LIN {X 0,Y 539.929,Z 932.451,A -85,B 0,C 180,E1 4064.865,E2 4064.865} C_VEL
LIN {X 0,Y 540.898,Z 908.583,A -85,B 0,C 180,E1 4068.356,E2 4068.356} C_VEL
LIN {X 0,Y 542.169,Z 880.394,A -85,B 0,C 180,E1 4071.395,E2 4071.395} C_VEL
LIN {X 0,Y 543.664,Z 848.735,A -85,B 0,C 180,E1 4073.926,E2 4073.926} C_VEL
LIN {X 0,Y 545.192,Z 813.47,A -85,B 0,C 180,E1 4075.928,E2 4075.928} C_VEL
LIN {X 0,Y 546.363,Z 778.099,A -85,B 0,C 180,E1 4077.245,E2 4077.245} C_VEL
LIN {X 0,Y 546.243,Z 753.317,A -85,B 0,C 180,E1 4077.845,E2 4077.845} C_VEL
LIN {X 0,Y 538.505,Z 733.66,A -85,B 0,C 180,E1 4078.65,E2 4078.65} C_VEL
LIN {X 0,Y 538.24,Z 733.66,A -85,B 0,C 180,E1 4084.237,E2 4084.237} C_VEL
LIN {X 0,Y 538.141,Z 733.66,A -85,B 0,C 180,E1 4090.325,E2 4090.325} C_VEL
LIN {X 0,Y 538.198,Z 733.66,A -85,B 0,C 180,E1 4095.304,E2 4095.304} C_VEL
LIN {X 0,Y 538.244,Z 733.66,A -85,B 0,C 180,E1 4101.765,E2 4101.765} C_VEL
LIN {X 0,Y 538.178,Z 733.66,A -85,B 0,C 180,E1 4107.685,E2 4107.685} C_VEL
LIN {X 0,Y 538.392,Z 733.66,A -85,B 0,C 180,E1 4113.256,E2 4113.256} C_VEL
LIN {X 0,Y 538.489,Z 733.66,A -85,B 0,C 180,E1 4118.557,E2 4118.557} C_VEL
LIN {X 0,Y 538.505,Z 733.66,A -85,B 0,C 180,E1 4123.667,E2 4123.667} C_VEL
LIN {X 0,Y 538.551,Z 733.66,A -85,B 0,C 180,E1 4130.286,E2 4130.286} C_VEL
LIN {X 0,Y 538.695,Z 733.66,A -85,B 0,C 180,E1 4135.16,E2 4135.16} C_VEL
LIN {X 0,Y 538.731,Z 733.66,A -85,B 0,C 180,E1 4139.996,E2 4139.996} C_VEL
LIN {X 0,Y 538.698,Z 733.66,A -85,B 0,C 180,E1 4144.833,E2 4144.833} C_VEL
LIN {X 0,Y 538.561,Z 733.66,A -85,B 0,C 180,E1 4150.268,E2 4150.268} C_VEL
LIN {X 0,Y 538.552,Z 733.66,A -85,B 0,C 180,E1 4154.652,E2 4154.652} C_VEL
LIN {X 0,Y 538.526,Z 733.66,A -85,B 0,C 180,E1 4159.713,E2 4159.713} C_VEL
LIN {X 0,Y 538.328,Z 733.66,A -85,B 0,C 180,E1 4165.302,E2 4165.302} C_VEL
LIN {X 0,Y 537.026,Z 733.66,A -85,B 0,C 180,E1 4166.225,E2 4166.225} C_VEL
LIN {X 0,Y 530.436,Z 733.66,A -85,B 0,C 180,E1 4168.737,E2 4168.737} C_VEL
LIN {X 0,Y 530.367,Z 733.66,A -85,B 0,C 180,E1 4168.975,E2 4168.975} C_VEL
LIN {X 0,Y 530.295,Z 733.66,A -85,B 0,C 180,E1 4174.816,E2 4174.816} C_VEL
LIN {X 0,Y 530.19,Z 733.66,A -85,B 0,C 180,E1 4181.05,E2 4181.05} C_VEL
LIN {X 0,Y 530.337,Z 733.66,A -85,B 0,C 180,E1 4186.749,E2 4186.749} C_VEL
LIN {X 0,Y 530.299,Z 733.66,A -85,B 0,C 180,E1 4193.067,E2 4193.067} C_VEL
LIN {X 0,Y 530.392,Z 734.199,A -85,B 0,C 180,E1 4198.178,E2 4198.178} C_VEL
LIN {X 0,Y 534.911,Z 747.208,A -85,B 0,C 180,E1 4199.252,E2 4199.252} C_VEL
LIN {X 0,Y 543.352,Z 759.578,A -85,B 0,C 180,E1 4200.686,E2 4200.686} C_VEL
LIN {X 0,Y 540.185,Z 771.164,A -85,B 0,C 180,E1 4201.27,E2 4201.27} C_VEL
LIN {X 0,Y 539.525,Z 822.398,A -85,B 0,C 180,E1 4202.164,E2 4202.164} C_VEL
LIN {X 0,Y 538.205,Z 858.389,A -85,B 0,C 180,E1 4203.418,E2 4203.418} C_VEL
LIN {X 0,Y 536.657,Z 892.998,A -85,B 0,C 180,E1 4205.297,E2 4205.297} C_VEL
LIN {X 0,Y 534.865,Z 926.522,A -85,B 0,C 180,E1 4207.881,E2 4207.881} C_VEL
LIN {X 0,Y 533.463,Z 953.726,A -85,B 0,C 180,E1 4210.734,E2 4210.734} C_VEL
LIN {X 0,Y 532.298,Z 977.994,A -85,B 0,C 180,E1 4214.111,E2 4214.111} C_VEL
LIN {X 0,Y 531.607,Z 996.677,A -85,B 0,C 180,E1 4217.666,E2 4217.666} C_VEL
LIN {X 0,Y 531.266,Z 1010.424,A -85,B 0,C 180,E1 4221.395,E2 4221.395} C_VEL
LIN {X 0,Y 531.098,Z 1018.952,A -85,B 0,C 180,E1 4225.093,E2 4225.093} C_VEL
LIN {X 0,Y 531.029,Z 1022.53,A -85,B 0,C 180,E1 4228.366,E2 4228.366} C_VEL
LIN {X 0,Y 531.093,Z 1022.529,A -85,B 0,C 180,E1 4231.633,E2 4231.633} C_VEL
LIN {X 0,Y 531.095,Z 1017.469,A -85,B 0,C 180,E1 4235.726,E2 4235.726} C_VEL
LIN {X 0,Y 531.28,Z 1007.861,A -85,B 0,C 180,E1 4239.431,E2 4239.431} C_VEL
LIN {X 0,Y 531.693,Z 992.833,A -85,B 0,C 180,E1 4243.168,E2 4243.168} C_VEL
LIN {X 0,Y 532.477,Z 971.655,A -85,B 0,C 180,E1 4246.872,E2 4246.872} C_VEL
LIN {X 0,Y 533.771,Z 946.485,A -85,B 0,C 180,E1 4250.107,E2 4250.107} C_VEL
LIN {X 0,Y 535.394,Z 917.124,A -85,B 0,C 180,E1 4252.931,E2 4252.931} C_VEL
LIN {X 0,Y 537.131,Z 884.48,A -85,B 0,C 180,E1 4255.23,E2 4255.23} C_VEL
LIN {X 0,Y 538.607,Z 850.059,A -85,B 0,C 180,E1 4256.929,E2 4256.929} C_VEL
LIN {X 0,Y 539.757,Z 813.547,A -85,B 0,C 180,E1 4258.047,E2 4258.047} C_VEL
LIN {X 0,Y 540.347,Z 770.37,A -85,B 0,C 180,E1 4258.776,E2 4258.776} C_VEL
LIN {X 0,Y 543.301,Z 759.584,A -85,B 0,C 180,E1 4259.319,E2 4259.319} C_VEL
LIN {X 0,Y 535.922,Z 748.545,A -85,B 0,C 180,E1 4260.605,E2 4260.605} C_VEL
LIN {X 0,Y 531.135,Z 737.856,A -85,B 0,C 180,E1 4261.416,E2 4261.416} C_VEL
LIN {X 0,Y 530.394,Z 733.66,A -85,B 0,C 180,E1 4261.772,E2 4261.772} C_VEL
LIN {X 0,Y 530.271,Z 733.66,A -85,B 0,C 180,E1 4266.929,E2 4266.929} C_VEL
LIN {X 0,Y 530.332,Z 733.66,A -85,B 0,C 180,E1 4273.251,E2 4273.251} C_VEL
LIN {X 0,Y 530.202,Z 733.66,A -85,B 0,C 180,E1 4278.951,E2 4278.951} C_VEL
LIN {X 0,Y 530.313,Z 733.66,A -85,B 0,C 180,E1 4285.185,E2 4285.185} C_VEL
LIN {X 0,Y 530.38,Z 733.66,A -85,B 0,C 180,E1 4290.974,E2 4290.974} C_VEL
LIN {X 0,Y 530.358,Z 733.66,A -85,B 0,C 180,E1 4296.447,E2 4296.447} C_VEL
LIN {X 0,Y 530.588,Z 733.66,A -85,B 0,C 180,E1 4299.925,E2 4299.925} C_VEL
LIN {X 0,Y 534.239,Z 751.767,A -85,B 0,C 180,E1 4300.375,E2 4300.375} C_VEL
LIN {X 0,Y 534.049,Z 781.281,A -85,B 0,C 180,E1 4301.36,E2 4301.36} C_VEL
LIN {X 0,Y 533.37,Z 807.505,A -85,B 0,C 180,E1 4302.911,E2 4302.911} C_VEL
LIN {X 0,Y 532.655,Z 830.205,A -85,B 0,C 180,E1 4304.993,E2 4304.993} C_VEL
LIN {X 0,Y 532.005,Z 848.565,A -85,B 0,C 180,E1 4307.471,E2 4307.471} C_VEL
LIN {X 0,Y 531.572,Z 861.83,A -85,B 0,C 180,E1 4310.164,E2 4310.164} C_VEL
LIN {X 0,Y 531.368,Z 871.236,A -85,B 0,C 180,E1 4313.459,E2 4313.459} C_VEL
LIN {X 0,Y 531.216,Z 874.4,A -85,B 0,C 180,E1 4316.736,E2 4316.736} C_VEL
LIN {X 0,Y 531.291,Z 871.871,A -85,B 0,C 180,E1 4320.004,E2 4320.004} C_VEL
LIN {X 0,Y 531.451,Z 864.702,A -85,B 0,C 180,E1 4322.861,E2 4322.861} C_VEL
LIN {X 0,Y 531.852,Z 850.948,A -85,B 0,C 180,E1 4325.927,E2 4325.927} C_VEL
LIN {X 0,Y 532.375,Z 832.207,A -85,B 0,C 180,E1 4328.59,E2 4328.59} C_VEL
LIN {X 0,Y 533.103,Z 809.618,A -85,B 0,C 180,E1 4330.745,E2 4330.745} C_VEL
LIN {X 0,Y 533.865,Z 783.985,A -85,B 0,C 180,E1 4332.354,E2 4332.354} C_VEL
LIN {X 0,Y 534.405,Z 755.268,A -85,B 0,C 180,E1 4333.417,E2 4333.417} C_VEL
LIN {X 0,Y 532.781,Z 741.992,A -85,B 0,C 180,E1 4333.748,E2 4333.748} C_VEL
LIN {X 0,Y 530.642,Z 733.66,A -85,B 0,C 180,E1 4334.04,E2 4334.04} C_VEL
LIN {X 0,Y 530.553,Z 733.66,A -85,B 0,C 180,E1 4340.029,E2 4340.029} C_VEL
LIN {X 0,Y 530.431,Z 733.66,A -85,B 0,C 180,E1 4345.354,E2 4345.354} C_VEL
LIN {X 0,Y 530.297,Z 733.66,A -85,B 0,C 180,E1 4351.069,E2 4351.069} C_VEL
LIN {X 0,Y 530.234,Z 733.66,A -85,B 0,C 180,E1 4356.914,E2 4356.914} C_VEL
LIN {X 0,Y 530.302,Z 733.66,A -85,B 0,C 180,E1 4363.256,E2 4363.256} C_VEL
LIN {X 0,Y 530.31,Z 733.66,A -85,B 0,C 180,E1 4368.954,E2 4368.954} C_VEL
LIN {X 0,Y 530.286,Z 733.66,A -85,B 0,C 180,E1 4375.177,E2 4375.177} C_VEL
LIN {X 0,Y 530.42,Z 733.66,A -85,B 0,C 180,E1 4380.828,E2 4380.828} C_VEL
LIN {X 0,Y 539.68,Z 758.857,A -85,B 0,C 180,E1 4381.801,E2 4381.801} C_VEL
LIN {X 0,Y 538.677,Z 797.066,A -85,B 0,C 180,E1 4382.911,E2 4382.911} C_VEL
LIN {X 0,Y 537.216,Z 832.111,A -85,B 0,C 180,E1 4384.59,E2 4384.59} C_VEL
LIN {X 0,Y 535.516,Z 864.375,A -85,B 0,C 180,E1 4386.8,E2 4386.8} C_VEL
LIN {X 0,Y 533.886,Z 895.221,A -85,B 0,C 180,E1 4389.706,E2 4389.706} C_VEL
LIN {X 0,Y 532.582,Z 920.869,A -85,B 0,C 180,E1 4392.968,E2 4392.968} C_VEL
LIN {X 0,Y 531.851,Z 941.307,A -85,B 0,C 180,E1 4396.474,E2 4396.474} C_VEL
LIN {X 0,Y 531.367,Z 956.651,A -85,B 0,C 180,E1 4400.156,E2 4400.156} C_VEL
LIN {X 0,Y 531.192,Z 965.865,A -85,B 0,C 180,E1 4403.453,E2 4403.453} C_VEL
LIN {X 0,Y 531.107,Z 971.214,A -85,B 0,C 180,E1 4406.732,E2 4406.732} C_VEL
LIN {X 0,Y 531.074,Z 972.997,A -85,B 0,C 180,E1 4410,E2 4410} C_VEL
LIN {X 0,Y 531.156,Z 970.398,A -85,B 0,C 180,E1 4413.883,E2 4413.883} C_VEL
LIN {X 0,Y 531.252,Z 962.625,A -85,B 0,C 180,E1 4417.781,E2 4417.781} C_VEL
LIN {X 0,Y 531.478,Z 950.035,A -85,B 0,C 180,E1 4421.503,E2 4421.503} C_VEL
LIN {X 0,Y 532.216,Z 931.471,A -85,B 0,C 180,E1 4425.257,E2 4425.257} C_VEL
LIN {X 0,Y 533.292,Z 906.861,A -85,B 0,C 180,E1 4428.842,E2 4428.842} C_VEL
LIN {X 0,Y 534.784,Z 878.331,A -85,B 0,C 180,E1 4431.905,E2 4431.905} C_VEL
LIN {X 0,Y 536.522,Z 845.585,A -85,B 0,C 180,E1 4434.487,E2 4434.487} C_VEL
LIN {X 0,Y 538.09,Z 813.068,A -85,B 0,C 180,E1 4436.316,E2 4436.316} C_VEL
LIN {X 0,Y 539.356,Z 778.111,A -85,B 0,C 180,E1 4437.629,E2 4437.629} C_VEL
LIN {X 0,Y 539.212,Z 755.599,A -85,B 0,C 180,E1 4438.198,E2 4438.198} C_VEL
LIN {X 0,Y 530.524,Z 733.66,A -85,B 0,C 180,E1 4439.114,E2 4439.114} C_VEL
LIN {X 0,Y 530.312,Z 733.66,A -85,B 0,C 180,E1 4444.822,E2 4444.822} C_VEL
LIN {X 0,Y 530.193,Z 733.66,A -85,B 0,C 180,E1 4451.058,E2 4451.058} C_VEL
LIN {X 0,Y 530.318,Z 733.66,A -85,B 0,C 180,E1 4456.745,E2 4456.745} C_VEL
LIN {X 0,Y 530.267,Z 733.66,A -85,B 0,C 180,E1 4463.155,E2 4463.155} C_VEL
LIN {X 0,Y 530.274,Z 733.66,A -85,B 0,C 180,E1 4469.07,E2 4469.07} C_VEL
LIN {X 0,Y 530.512,Z 733.66,A -85,B 0,C 180,E1 4474.65,E2 4474.65} C_VEL
LIN {X 0,Y 530.696,Z 733.66,A -85,B 0,C 180,E1 4480.306,E2 4480.306} C_VEL
LIN {X 0,Y 530.363,Z 733.66,A -85,B 0,C 180,E1 4486.083,E2 4486.083} C_VEL
LIN {X 0,Y 530.653,Z 733.66,A -85,B 0,C 180,E1 4491.795,E2 4491.795} C_VEL
LIN {X 0,Y 530.732,Z 733.66,A -85,B 0,C 180,E1 4496.86,E2 4496.86} C_VEL
LIN {X 0,Y 530.746,Z 733.66,A -85,B 0,C 180,E1 4501.631,E2 4501.631} C_VEL
LIN {X 0,Y 530.702,Z 733.66,A -85,B 0,C 180,E1 4506.549,E2 4506.549} C_VEL
LIN {X 0,Y 530.651,Z 733.66,A -85,B 0,C 180,E1 4511.517,E2 4511.517} C_VEL
LIN {X 0,Y 530.598,Z 733.66,A -85,B 0,C 180,E1 4516.575,E2 4516.575} C_VEL
LIN {X 0,Y 530.538,Z 733.66,A -85,B 0,C 180,E1 4521.772,E2 4521.772} C_VEL
LIN {X 0,Y 530.358,Z 733.66,A -85,B 0,C 180,E1 4527.747,E2 4527.747} C_VEL
LIN {X 0,Y 530.367,Z 733.66,A -85,B 0,C 180,E1 4528.975,E2 4528.975} C_VEL
LIN {X 0,Y 527.852,Z 733.66,A -85,B 0,C 180,E1 4530.369,E2 4530.369} C_VEL
LIN {X 0,Y 522.463,Z 733.66,A -85,B 0,C 180,E1 4532.458,E2 4532.458} C_VEL
LIN {X 0,Y 522.395,Z 733.66,A -85,B 0,C 180,E1 4532.699,E2 4532.699} C_VEL
LIN {X 0,Y 522.248,Z 733.66,A -85,B 0,C 180,E1 4538.484,E2 4538.484} C_VEL
LIN {X 0,Y 522.388,Z 733.66,A -85,B 0,C 180,E1 4544.068,E2 4544.068} C_VEL
LIN {X 0,Y 522.41,Z 733.66,A -85,B 0,C 180,E1 4550.385,E2 4550.385} C_VEL
LIN {X 0,Y 522.363,Z 733.66,A -85,B 0,C 180,E1 4556.583,E2 4556.583} C_VEL
LIN {X 0,Y 522.469,Z 734.17,A -85,B 0,C 180,E1 4557.761,E2 4557.761} C_VEL
LIN {X 0,Y 528.528,Z 751.834,A -85,B 0,C 180,E1 4559.239,E2 4559.239} C_VEL
LIN {X 0,Y 536.281,Z 762.43,A -85,B 0,C 180,E1 4560.311,E2 4560.311} C_VEL
LIN {X 0,Y 533.224,Z 774.555,A -85,B 0,C 180,E1 4560.915,E2 4560.915} C_VEL
LIN {X 0,Y 532.534,Z 822.756,A -85,B 0,C 180,E1 4561.776,E2 4561.776} C_VEL
LIN {X 0,Y 531.071,Z 859.288,A -85,B 0,C 180,E1 4563.075,E2 4563.075} C_VEL
LIN {X 0,Y 529.28,Z 894.607,A -85,B 0,C 180,E1 4565.042,E2 4565.042} C_VEL
LIN {X 0,Y 527.318,Z 927.968,A -85,B 0,C 180,E1 4567.683,E2 4567.683} C_VEL
LIN {X 0,Y 525.636,Z 957.199,A -85,B 0,C 180,E1 4570.873,E2 4570.873} C_VEL
LIN {X 0,Y 524.433,Z 980.46,A -85,B 0,C 180,E1 4574.296,E2 4574.296} C_VEL
LIN {X 0,Y 523.674,Z 998.511,A -85,B 0,C 180,E1 4577.9,E2 4577.9} C_VEL
LIN {X 0,Y 523.342,Z 1011.603,A -85,B 0,C 180,E1 4581.682,E2 4581.682} C_VEL
LIN {X 0,Y 523.201,Z 1018.949,A -85,B 0,C 180,E1 4585.019,E2 4585.019} C_VEL
LIN {X 0,Y 523.144,Z 1022.532,A -85,B 0,C 180,E1 4588.341,E2 4588.341} C_VEL
LIN {X 0,Y 523.204,Z 1022.531,A -85,B 0,C 180,E1 4591.658,E2 4591.658} C_VEL
LIN {X 0,Y 523.21,Z 1017.471,A -85,B 0,C 180,E1 4595.813,E2 4595.813} C_VEL
LIN {X 0,Y 523.411,Z 1007.857,A -85,B 0,C 180,E1 4599.574,E2 4599.574} C_VEL
LIN {X 0,Y 523.869,Z 992.835,A -85,B 0,C 180,E1 4603.368,E2 4603.368} C_VEL
LIN {X 0,Y 524.758,Z 972.047,A -85,B 0,C 180,E1 4607.066,E2 4607.066} C_VEL
LIN {X 0,Y 526.17,Z 946.886,A -85,B 0,C 180,E1 4610.364,E2 4610.364} C_VEL
LIN {X 0,Y 528.004,Z 917.072,A -85,B 0,C 180,E1 4613.275,E2 4613.275} C_VEL
LIN {X 0,Y 529.888,Z 884.475,A -85,B 0,C 180,E1 4615.6,E2 4615.6} C_VEL
LIN {X 0,Y 531.544,Z 849.967,A -85,B 0,C 180,E1 4617.32,E2 4617.32} C_VEL
LIN {X 0,Y 532.802,Z 813.504,A -85,B 0,C 180,E1 4618.448,E2 4618.448} C_VEL
LIN {X 0,Y 533.558,Z 772.405,A -85,B 0,C 180,E1 4619.177,E2 4619.177} C_VEL
LIN {X 0,Y 535.699,Z 761.602,A -85,B 0,C 180,E1 4619.779,E2 4619.779} C_VEL
LIN {X 0,Y 525.526,Z 746.23,A -85,B 0,C 180,E1 4621.098,E2 4621.098} C_VEL
LIN {X 0,Y 522.474,Z 733.66,A -85,B 0,C 180,E1 4622.031,E2 4622.031} C_VEL
LIN {X 0,Y 522.332,Z 733.66,A -85,B 0,C 180,E1 4628.506,E2 4628.506} C_VEL
LIN {X 0,Y 522.41,Z 733.66,A -85,B 0,C 180,E1 4634.074,E2 4634.074} C_VEL
LIN {X 0,Y 522.299,Z 733.66,A -85,B 0,C 180,E1 4640.383,E2 4640.383} C_VEL
LIN {X 0,Y 522.441,Z 733.66,A -85,B 0,C 180,E1 4646.596,E2 4646.596} C_VEL
LIN {X 0,Y 522.393,Z 733.66,A -85,B 0,C 180,E1 4652.377,E2 4652.377} C_VEL
LIN {X 0,Y 522.501,Z 733.66,A -85,B 0,C 180,E1 4658.016,E2 4658.016} C_VEL
LIN {X 0,Y 522.642,Z 734.005,A -85,B 0,C 180,E1 4659.662,E2 4659.662} C_VEL
LIN {X 0,Y 526.784,Z 753.759,A -85,B 0,C 180,E1 4660.154,E2 4660.154} C_VEL
LIN {X 0,Y 526.518,Z 782.775,A -85,B 0,C 180,E1 4661.142,E2 4661.142} C_VEL
LIN {X 0,Y 525.827,Z 808.359,A -85,B 0,C 180,E1 4662.67,E2 4662.67} C_VEL
LIN {X 0,Y 525.1,Z 830.995,A -85,B 0,C 180,E1 4664.75,E2 4664.75} C_VEL
LIN {X 0,Y 524.365,Z 849.627,A -85,B 0,C 180,E1 4667.285,E2 4667.285} C_VEL
LIN {X 0,Y 523.869,Z 862.972,A -85,B 0,C 180,E1 4670.018,E2 4670.018} C_VEL
LIN {X 0,Y 523.711,Z 870.701,A -85,B 0,C 180,E1 4672.529,E2 4672.529} C_VEL
LIN {X 0,Y 523.586,Z 874.779,A -85,B 0,C 180,E1 4675.027,E2 4675.027} C_VEL
LIN {X 0,Y 523.461,Z 875.097,A -85,B 0,C 180,E1 4678.346,E2 4678.346} C_VEL
LIN {X 0,Y 523.546,Z 869.653,A -85,B 0,C 180,E1 4681.661,E2 4681.661} C_VEL
LIN {X 0,Y 523.874,Z 859.139,A -85,B 0,C 180,E1 4684.648,E2 4684.648} C_VEL
LIN {X 0,Y 524.375,Z 843.193,A -85,B 0,C 180,E1 4687.469,E2 4687.469} C_VEL
LIN {X 0,Y 525.111,Z 821.857,A -85,B 0,C 180,E1 4689.966,E2 4689.966} C_VEL
LIN {X 0,Y 525.957,Z 796.971,A -85,B 0,C 180,E1 4691.901,E2 4691.901} C_VEL
LIN {X 0,Y 526.575,Z 769.577,A -85,B 0,C 180,E1 4693.244,E2 4693.244} C_VEL
LIN {X 0,Y 526.194,Z 746.991,A -85,B 0,C 180,E1 4693.888,E2 4693.888} C_VEL
LIN {X 0,Y 522.705,Z 733.66,A -85,B 0,C 180,E1 4694.258,E2 4694.258} C_VEL
LIN {X 0,Y 522.614,Z 733.66,A -85,B 0,C 180,E1 4700.347,E2 4700.347} C_VEL
LIN {X 0,Y 522.434,Z 733.66,A -85,B 0,C 180,E1 4706.048,E2 4706.048} C_VEL
LIN {X 0,Y 522.367,Z 733.66,A -85,B 0,C 180,E1 4711.451,E2 4711.451} C_VEL
LIN {X 0,Y 522.277,Z 733.66,A -85,B 0,C 180,E1 4717.505,E2 4717.505} C_VEL
LIN {X 0,Y 522.382,Z 733.66,A -85,B 0,C 180,E1 4723.564,E2 4723.564} C_VEL
LIN {X 0,Y 522.436,Z 733.66,A -85,B 0,C 180,E1 4728.898,E2 4728.898} C_VEL
LIN {X 0,Y 522.316,Z 733.66,A -85,B 0,C 180,E1 4734.567,E2 4734.567} C_VEL
LIN {X 0,Y 522.472,Z 733.66,A -85,B 0,C 180,E1 4740.322,E2 4740.322} C_VEL
LIN {X 0,Y 532.696,Z 761.121,A -85,B 0,C 180,E1 4741.446,E2 4741.446} C_VEL
LIN {X 0,Y 531.529,Z 799.009,A -85,B 0,C 180,E1 4742.6,E2 4742.6} C_VEL
LIN {X 0,Y 529.903,Z 833.765,A -85,B 0,C 180,E1 4744.316,E2 4744.316} C_VEL
LIN {X 0,Y 527.982,Z 866.735,A -85,B 0,C 180,E1 4746.647,E2 4746.647} C_VEL
LIN {X 0,Y 526.281,Z 895.955,A -85,B 0,C 180,E1 4749.485,E2 4749.485} C_VEL
LIN {X 0,Y 524.901,Z 920.495,A -85,B 0,C 180,E1 4752.656,E2 4752.656} C_VEL
LIN {X 0,Y 524.042,Z 941.496,A -85,B 0,C 180,E1 4756.307,E2 4756.307} C_VEL
LIN {X 0,Y 523.496,Z 956.649,A -85,B 0,C 180,E1 4760.007,E2 4760.007} C_VEL
LIN {X 0,Y 523.293,Z 965.864,A -85,B 0,C 180,E1 4763.354,E2 4763.354} C_VEL
LIN {X 0,Y 523.219,Z 971.213,A -85,B 0,C 180,E1 4766.682,E2 4766.682} C_VEL
LIN {X 0,Y 523.184,Z 972.997,A -85,B 0,C 180,E1 4770,E2 4770} C_VEL
LIN {X 0,Y 523.248,Z 970.399,A -85,B 0,C 180,E1 4773.942,E2 4773.942} C_VEL
LIN {X 0,Y 523.364,Z 962.627,A -85,B 0,C 180,E1 4777.899,E2 4777.899} C_VEL
LIN {X 0,Y 523.612,Z 950.036,A -85,B 0,C 180,E1 4781.678,E2 4781.678} C_VEL
LIN {X 0,Y 524.414,Z 931.478,A -85,B 0,C 180,E1 4785.49,E2 4785.49} C_VEL
LIN {X 0,Y 525.662,Z 906.864,A -85,B 0,C 180,E1 4789.126,E2 4789.126} C_VEL
LIN {X 0,Y 527.234,Z 879.552,A -85,B 0,C 180,E1 4792.116,E2 4792.116} C_VEL
LIN {X 0,Y 529.145,Z 847.228,A -85,B 0,C 180,E1 4794.739,E2 4794.739} C_VEL
LIN {X 0,Y 530.988,Z 813.08,A -85,B 0,C 180,E1 4796.695,E2 4796.695} C_VEL
LIN {X 0,Y 532.325,Z 778.628,A -85,B 0,C 180,E1 4798.01,E2 4798.01} C_VEL
LIN {X 0,Y 532.064,Z 757.239,A -85,B 0,C 180,E1 4798.58,E2 4798.58} C_VEL
LIN {X 0,Y 522.551,Z 733.66,A -85,B 0,C 180,E1 4799.626,E2 4799.626} C_VEL
LIN {X 0,Y 522.315,Z 733.66,A -85,B 0,C 180,E1 4805.739,E2 4805.739} C_VEL
LIN {X 0,Y 522.303,Z 733.66,A -85,B 0,C 180,E1 4811.816,E2 4811.816} C_VEL
LIN {X 0,Y 522.371,Z 733.66,A -85,B 0,C 180,E1 4818.188,E2 4818.188} C_VEL
LIN {X 0,Y 522.302,Z 733.66,A -85,B 0,C 180,E1 4824.563,E2 4824.563} C_VEL
LIN {X 0,Y 522.375,Z 733.66,A -85,B 0,C 180,E1 4830.477,E2 4830.477} C_VEL
LIN {X 0,Y 522.594,Z 733.66,A -85,B 0,C 180,E1 4836.068,E2 4836.068} C_VEL
LIN {X 0,Y 522.74,Z 733.66,A -85,B 0,C 180,E1 4841.418,E2 4841.418} C_VEL
LIN {X 0,Y 522.626,Z 733.66,A -85,B 0,C 180,E1 4848.296,E2 4848.296} C_VEL
LIN {X 0,Y 522.94,Z 733.66,A -85,B 0,C 180,E1 4853.346,E2 4853.346} C_VEL
LIN {X 0,Y 522.949,Z 733.66,A -85,B 0,C 180,E1 4859.996,E2 4859.996} C_VEL
LIN {X 0,Y 522.87,Z 733.66,A -85,B 0,C 180,E1 4864.98,E2 4864.98} C_VEL
LIN {X 0,Y 522.808,Z 733.66,A -85,B 0,C 180,E1 4870.045,E2 4870.045} C_VEL
LIN {X 0,Y 522.703,Z 733.66,A -85,B 0,C 180,E1 4875.107,E2 4875.107} C_VEL
LIN {X 0,Y 522.632,Z 733.66,A -85,B 0,C 180,E1 4880.338,E2 4880.338} C_VEL
LIN {X 0,Y 522.463,Z 733.66,A -85,B 0,C 180,E1 4886.054,E2 4886.054} C_VEL
LIN {X 0,Y 522.369,Z 733.66,A -85,B 0,C 180,E1 4891.442,E2 4891.442} C_VEL
LIN {X 0,Y 522.395,Z 733.66,A -85,B 0,C 180,E1 4892.699,E2 4892.699} C_VEL
LIN {X 0,Y 519.924,Z 733.66,A -85,B 0,C 180,E1 4894.111,E2 4894.111} C_VEL
LIN {X 0,Y 514.447,Z 733.66,A -85,B 0,C 180,E1 4896.226,E2 4896.226} C_VEL
LIN {X 0,Y 514.339,Z 733.66,A -85,B 0,C 180,E1 4896.471,E2 4896.471} C_VEL
LIN {X 0,Y 514.412,Z 733.66,A -85,B 0,C 180,E1 4902.622,E2 4902.622} C_VEL
LIN {X 0,Y 514.482,Z 733.66,A -85,B 0,C 180,E1 4907.4,E2 4907.4} C_VEL
LIN {X 0,Y 514.453,Z 733.66,A -85,B 0,C 180,E1 4912.611,E2 4912.611} C_VEL
LIN {X 0,Y 514.499,Z 733.748,A -85,B 0,C 180,E1 4917.299,E2 4917.299} C_VEL
LIN {X 0,Y 521.232,Z 755.025,A -85,B 0,C 180,E1 4919.085,E2 4919.085} C_VEL
LIN {X 0,Y 528.098,Z 766.006,A -85,B 0,C 180,E1 4920.141,E2 4920.141} C_VEL
LIN {X 0,Y 526.137,Z 775.03,A -85,B 0,C 180,E1 4920.548,E2 4920.548} C_VEL
LIN {X 0,Y 525.43,Z 822.995,A -85,B 0,C 180,E1 4921.403,E2 4921.403} C_VEL
LIN {X 0,Y 523.929,Z 860.182,A -85,B 0,C 180,E1 4922.723,E2 4922.723} C_VEL
LIN {X 0,Y 521.922,Z 896.215,A -85,B 0,C 180,E1 4924.78,E2 4924.78} C_VEL
LIN {X 0,Y 519.855,Z 928.496,A -85,B 0,C 180,E1 4927.396,E2 4927.396} C_VEL
LIN {X 0,Y 518.038,Z 957.195,A -85,B 0,C 180,E1 4930.581,E2 4930.581} C_VEL
LIN {X 0,Y 516.671,Z 980.455,A -85,B 0,C 180,E1 4934.054,E2 4934.054} C_VEL
LIN {X 0,Y 515.868,Z 998.515,A -85,B 0,C 180,E1 4937.714,E2 4937.714} C_VEL
LIN {X 0,Y 515.479,Z 1012.764,A -85,B 0,C 180,E1 4941.98,E2 4941.98} C_VEL
LIN {X 0,Y 515.301,Z 1020.165,A -85,B 0,C 180,E1 4945.787,E2 4945.787} C_VEL
LIN {X 0,Y 515.229,Z 1023,A -85,B 0,C 180,E1 4950,E2 4950} C_VEL
LIN {X 0,Y 515.364,Z 1020.171,A -85,B 0,C 180,E1 4954.212,E2 4954.212} C_VEL
LIN {X 0,Y 515.511,Z 1011.596,A -85,B 0,C 180,E1 4958.444,E2 4958.444} C_VEL
LIN {X 0,Y 515.879,Z 998.519,A -85,B 0,C 180,E1 4962.285,E2 4962.285} C_VEL
LIN {X 0,Y 516.78,Z 977.997,A -85,B 0,C 180,E1 4966.379,E2 4966.379} C_VEL
LIN {X 0,Y 518.204,Z 953.723,A -85,B 0,C 180,E1 4969.856,E2 4969.856} C_VEL
LIN {X 0,Y 520.078,Z 924.83,A -85,B 0,C 180,E1 4972.943,E2 4972.943} C_VEL
LIN {X 0,Y 522.195,Z 892.994,A -85,B 0,C 180,E1 4975.435,E2 4975.435} C_VEL
LIN {X 0,Y 524.05,Z 858.372,A -85,B 0,C 180,E1 4977.36,E2 4977.36} C_VEL
LIN {X 0,Y 525.319,Z 821.778,A -85,B 0,C 180,E1 4978.622,E2 4978.622} C_VEL
LIN {X 0,Y 526.33,Z 771.816,A -85,B 0,C 180,E1 4979.512,E2 4979.512} C_VEL
LIN {X 0,Y 527.445,Z 764.055,A -85,B 0,C 180,E1 4979.948,E2 4979.948} C_VEL
LIN {X 0,Y 517.749,Z 747.778,A -85,B 0,C 180,E1 4981.27,E2 4981.27} C_VEL
LIN {X 0,Y 514.544,Z 733.66,A -85,B 0,C 180,E1 4982.314,E2 4982.314} C_VEL
LIN {X 0,Y 514.413,Z 733.66,A -85,B 0,C 180,E1 4988.177,E2 4988.177} C_VEL
LIN {X 0,Y 514.479,Z 733.66,A -85,B 0,C 180,E1 4992.639,E2 4992.639} C_VEL
LIN {X 0,Y 514.409,Z 733.66,A -85,B 0,C 180,E1 4997.4,E2 4997.4} C_VEL
LIN {X 0,Y 514.392,Z 733.66,A -85,B 0,C 180,E1 5003.943,E2 5003.943} C_VEL
LIN {X 0,Y 514.501,Z 733.66,A -85,B 0,C 180,E1 5009.988,E2 5009.988} C_VEL
LIN {X 0,Y 514.543,Z 733.66,A -85,B 0,C 180,E1 5015.811,E2 5015.811} C_VEL
LIN {X 0,Y 514.701,Z 733.66,A -85,B 0,C 180,E1 5019.334,E2 5019.334} C_VEL
LIN {X 0,Y 519.331,Z 755.199,A -85,B 0,C 180,E1 5019.91,E2 5019.91} C_VEL
LIN {X 0,Y 519.046,Z 783.644,A -85,B 0,C 180,E1 5020.888,E2 5020.888} C_VEL
LIN {X 0,Y 518.283,Z 810.245,A -85,B 0,C 180,E1 5022.5,E2 5022.5} C_VEL
LIN {X 0,Y 517.545,Z 831.941,A -85,B 0,C 180,E1 5024.522,E2 5024.522} C_VEL
LIN {X 0,Y 516.73,Z 850.685,A -85,B 0,C 180,E1 5027.094,E2 5027.094} C_VEL
LIN {X 0,Y 516.144,Z 864.117,A -85,B 0,C 180,E1 5029.867,E2 5029.867} C_VEL
LIN {X 0,Y 515.964,Z 871.908,A -85,B 0,C 180,E1 5032.416,E2 5032.416} C_VEL
LIN {X 0,Y 515.806,Z 876.009,A -85,B 0,C 180,E1 5034.952,E2 5034.952} C_VEL
LIN {X 0,Y 515.674,Z 876.371,A -85,B 0,C 180,E1 5038.321,E2 5038.321} C_VEL
LIN {X 0,Y 515.767,Z 870.936,A -85,B 0,C 180,E1 5041.686,E2 5041.686} C_VEL
LIN {X 0,Y 516.131,Z 860.143,A -85,B 0,C 180,E1 5044.786,E2 5044.786} C_VEL
LIN {X 0,Y 516.674,Z 844.526,A -85,B 0,C 180,E1 5047.581,E2 5047.581} C_VEL
LIN {X 0,Y 517.474,Z 823.307,A -85,B 0,C 180,E1 5050.114,E2 5050.114} C_VEL
LIN {X 0,Y 518.364,Z 798.25,A -85,B 0,C 180,E1 5052.099,E2 5052.099} C_VEL
LIN {X 0,Y 519.047,Z 770.146,A -85,B 0,C 180,E1 5053.498,E2 5053.498} C_VEL
LIN {X 0,Y 518.556,Z 747.98,A -85,B 0,C 180,E1 5054.142,E2 5054.142} C_VEL
LIN {X 0,Y 514.779,Z 733.66,A -85,B 0,C 180,E1 5054.52,E2 5054.52} C_VEL
LIN {X 0,Y 514.681,Z 733.66,A -85,B 0,C 180,E1 5060.675,E2 5060.675} C_VEL
LIN {X 0,Y 514.531,Z 733.66,A -85,B 0,C 180,E1 5066.196,E2 5066.196} C_VEL
LIN {X 0,Y 514.453,Z 733.66,A -85,B 0,C 180,E1 5071.992,E2 5071.992} C_VEL
LIN {X 0,Y 514.354,Z 733.66,A -85,B 0,C 180,E1 5078.185,E2 5078.185} C_VEL
LIN {X 0,Y 514.404,Z 733.66,A -85,B 0,C 180,E1 5082.621,E2 5082.621} C_VEL
LIN {X 0,Y 514.477,Z 733.66,A -85,B 0,C 180,E1 5087.4,E2 5087.4} C_VEL
LIN {X 0,Y 514.415,Z 733.66,A -85,B 0,C 180,E1 5092.629,E2 5092.629} C_VEL
LIN {X 0,Y 514.445,Z 733.66,A -85,B 0,C 180,E1 5098.598,E2 5098.598} C_VEL
LIN {X 0,Y 514.518,Z 733.66,A -85,B 0,C 180,E1 5099.811,E2 5099.811} C_VEL
LIN {X 0,Y 525.717,Z 763.32,A -85,B 0,C 180,E1 5101.082,E2 5101.082} C_VEL
LIN {X 0,Y 524.43,Z 800.196,A -85,B 0,C 180,E1 5102.246,E2 5102.246} C_VEL
LIN {X 0,Y 522.547,Z 836.512,A -85,B 0,C 180,E1 5104.099,E2 5104.099} C_VEL
LIN {X 0,Y 520.405,Z 869.947,A -85,B 0,C 180,E1 5106.58,E2 5106.58} C_VEL
LIN {X 0,Y 518.53,Z 898.692,A -85,B 0,C 180,E1 5109.489,E2 5109.489} C_VEL
LIN {X 0,Y 516.976,Z 924.274,A -85,B 0,C 180,E1 5112.97,E2 5112.97} C_VEL
LIN {X 0,Y 516.042,Z 944.977,A -85,B 0,C 180,E1 5116.857,E2 5116.857} C_VEL
LIN {X 0,Y 515.542,Z 959.309,A -85,B 0,C 180,E1 5120.705,E2 5120.705} C_VEL
LIN {X 0,Y 515.287,Z 969.034,A -85,B 0,C 180,E1 5124.943,E2 5124.943} C_VEL
LIN {X 0,Y 515.246,Z 972.536,A -85,B 0,C 180,E1 5128.316,E2 5128.316} C_VEL
LIN {X 0,Y 515.265,Z 972.021,A -85,B 0,C 180,E1 5132.444,E2 5132.444} C_VEL
LIN {X 0,Y 515.388,Z 965.659,A -85,B 0,C 180,E1 5136.749,E2 5136.749} C_VEL
LIN {X 0,Y 515.661,Z 954.617,A -85,B 0,C 180,E1 5140.639,E2 5140.639} C_VEL
LIN {X 0,Y 516.382,Z 937.46,A -85,B 0,C 180,E1 5144.622,E2 5144.622} C_VEL
LIN {X 0,Y 517.586,Z 914.425,A -85,B 0,C 180,E1 5148.405,E2 5148.405} C_VEL
LIN {X 0,Y 519.328,Z 887.037,A -85,B 0,C 180,E1 5151.704,E2 5151.704} C_VEL
LIN {X 0,Y 521.307,Z 856.29,A -85,B 0,C 180,E1 5154.449,E2 5154.449} C_VEL
LIN {X 0,Y 523.264,Z 822.709,A -85,B 0,C 180,E1 5156.604,E2 5156.604} C_VEL
LIN {X 0,Y 524.994,Z 786.31,A -85,B 0,C 180,E1 5158.185,E2 5158.185} C_VEL
LIN {X 0,Y 525.405,Z 760.309,A -85,B 0,C 180,E1 5158.921,E2 5158.921} C_VEL
LIN {X 0,Y 514.55,Z 733.66,A -85,B 0,C 180,E1 5160.134,E2 5160.134} C_VEL
LIN {X 0,Y 514.397,Z 733.66,A -85,B 0,C 180,E1 5166.064,E2 5166.064} C_VEL
LIN {X 0,Y 514.37,Z 733.66,A -85,B 0,C 180,E1 5170.36,E2 5170.36} C_VEL
LIN {X 0,Y 514.378,Z 733.66,A -85,B 0,C 180,E1 5175.051,E2 5175.051} C_VEL
LIN {X 0,Y 514.439,Z 733.66,A -85,B 0,C 180,E1 5179.928,E2 5179.928} C_VEL
LIN {X 0,Y 514.372,Z 733.66,A -85,B 0,C 180,E1 5185.992,E2 5185.992} C_VEL
LIN {X 0,Y 514.532,Z 733.66,A -85,B 0,C 180,E1 5191.982,E2 5191.982} C_VEL
LIN {X 0,Y 514.68,Z 733.66,A -85,B 0,C 180,E1 5197.513,E2 5197.513} C_VEL
LIN {X 0,Y 514.781,Z 733.66,A -85,B 0,C 180,E1 5202.892,E2 5202.892} C_VEL
LIN {X 0,Y 514.788,Z 733.66,A -85,B 0,C 180,E1 5209.832,E2 5209.832} C_VEL
LIN {X 0,Y 514.986,Z 733.66,A -85,B 0,C 180,E1 5214.936,E2 5214.936} C_VEL
LIN {X 0,Y 515.048,Z 733.66,A -85,B 0,C 180,E1 5219.996,E2 5219.996} C_VEL
LIN {X 0,Y 514.965,Z 733.66,A -85,B 0,C 180,E1 5225.056,E2 5225.056} C_VEL
LIN {X 0,Y 514.916,Z 733.66,A -85,B 0,C 180,E1 5230.157,E2 5230.157} C_VEL
LIN {X 0,Y 514.792,Z 733.66,A -85,B 0,C 180,E1 5235.345,E2 5235.345} C_VEL
LIN {X 0,Y 514.695,Z 733.66,A -85,B 0,C 180,E1 5240.666,E2 5240.666} C_VEL
LIN {X 0,Y 514.56,Z 733.66,A -85,B 0,C 180,E1 5246.186,E2 5246.186} C_VEL
LIN {X 0,Y 514.48,Z 733.66,A -85,B 0,C 180,E1 5251.981,E2 5251.981} C_VEL
LIN {X 0,Y 514.339,Z 733.66,A -85,B 0,C 180,E1 5256.471,E2 5256.471} C_VEL
LIN {X 0,Y 513.028,Z 733.66,A -85,B 0,C 180,E1 5257.437,E2 5257.437} C_VEL
LIN {X 0,Y 506.395,Z 733.66,A -85,B 0,C 180,E1 5260.069,E2 5260.069} C_VEL
LIN {X 0,Y 506.313,Z 733.66,A -85,B 0,C 180,E1 5260.319,E2 5260.319} C_VEL
LIN {X 0,Y 506.495,Z 733.66,A -85,B 0,C 180,E1 5266.563,E2 5266.563} C_VEL
LIN {X 0,Y 506.52,Z 733.66,A -85,B 0,C 180,E1 5273.284,E2 5273.284} C_VEL
LIN {X 0,Y 506.593,Z 734.161,A -85,B 0,C 180,E1 5276.865,E2 5276.865} C_VEL
LIN {X 0,Y 514.132,Z 758.461,A -85,B 0,C 180,E1 5278.954,E2 5278.954} C_VEL
LIN {X 0,Y 520.152,Z 768.39,A -85,B 0,C 180,E1 5279.916,E2 5279.916} C_VEL
LIN {X 0,Y 519.012,Z 777.383,A -85,B 0,C 180,E1 5280.202,E2 5280.202} C_VEL
LIN {X 0,Y 518.155,Z 823.607,A -85,B 0,C 180,E1 5281.07,E2 5281.07} C_VEL
LIN {X 0,Y 516.532,Z 861.273,A -85,B 0,C 180,E1 5282.445,E2 5282.445} C_VEL
LIN {X 0,Y 514.686,Z 896.1,A -85,B 0,C 180,E1 5284.4,E2 5284.4} C_VEL
LIN {X 0,Y 512.531,Z 927.162,A -85,B 0,C 180,E1 5286.926,E2 5286.926} C_VEL
LIN {X 0,Y 510.554,Z 955.451,A -85,B 0,C 180,E1 5290.059,E2 5290.059} C_VEL
LIN {X 0,Y 508.983,Z 979.216,A -85,B 0,C 180,E1 5293.584,E2 5293.584} C_VEL
LIN {X 0,Y 508.037,Z 998.518,A -85,B 0,C 180,E1 5297.521,E2 5297.521} C_VEL
LIN {X 0,Y 507.586,Z 1012.765,A -85,B 0,C 180,E1 5301.854,E2 5301.854} C_VEL
LIN {X 0,Y 507.399,Z 1020.161,A -85,B 0,C 180,E1 5305.721,E2 5305.721} C_VEL
LIN {X 0,Y 507.341,Z 1023,A -85,B 0,C 180,E1 5310,E2 5310} C_VEL
LIN {X 0,Y 507.464,Z 1020.166,A -85,B 0,C 180,E1 5314.277,E2 5314.277} C_VEL
LIN {X 0,Y 507.616,Z 1011.592,A -85,B 0,C 180,E1 5318.577,E2 5318.577} C_VEL
LIN {X 0,Y 508.028,Z 998.523,A -85,B 0,C 180,E1 5322.478,E2 5322.478} C_VEL
LIN {X 0,Y 509.019,Z 977.993,A -85,B 0,C 180,E1 5326.636,E2 5326.636} C_VEL
LIN {X 0,Y 510.598,Z 953.718,A -85,B 0,C 180,E1 5330.164,E2 5330.164} C_VEL
LIN {X 0,Y 512.616,Z 925.483,A -85,B 0,C 180,E1 5333.233,E2 5333.233} C_VEL
LIN {X 0,Y 514.842,Z 894.457,A -85,B 0,C 180,E1 5335.707,E2 5335.707} C_VEL
LIN {X 0,Y 516.464,Z 860.348,A -85,B 0,C 180,E1 5337.558,E2 5337.558} C_VEL
LIN {X 0,Y 517.899,Z 821.255,A -85,B 0,C 180,E1 5338.915,E2 5338.915} C_VEL
LIN {X 0,Y 519.115,Z 770.112,A -85,B 0,C 180,E1 5339.844,E2 5339.844} C_VEL
LIN {X 0,Y 519.412,Z 766.388,A -85,B 0,C 180,E1 5340.064,E2 5340.064} C_VEL
LIN {X 0,Y 510.779,Z 751.59,A -85,B 0,C 180,E1 5341.275,E2 5341.275} C_VEL
LIN {X 0,Y 506.65,Z 733.66,A -85,B 0,C 180,E1 5342.623,E2 5342.623} C_VEL
LIN {X 0,Y 506.475,Z 733.66,A -85,B 0,C 180,E1 5348.999,E2 5348.999} C_VEL
LIN {X 0,Y 506.464,Z 733.66,A -85,B 0,C 180,E1 5354.161,E2 5354.161} C_VEL
LIN {X 0,Y 506.408,Z 733.66,A -85,B 0,C 180,E1 5358.878,E2 5358.878} C_VEL
LIN {X 0,Y 506.506,Z 733.66,A -85,B 0,C 180,E1 5365.398,E2 5365.398} C_VEL
LIN {X 0,Y 506.509,Z 733.66,A -85,B 0,C 180,E1 5371.433,E2 5371.433} C_VEL
LIN {X 0,Y 506.662,Z 733.66,A -85,B 0,C 180,E1 5377.879,E2 5377.879} C_VEL
LIN {X 0,Y 506.732,Z 733.66,A -85,B 0,C 180,E1 5378.994,E2 5378.994} C_VEL
LIN {X 0,Y 511.795,Z 754.605,A -85,B 0,C 180,E1 5379.613,E2 5379.613} C_VEL
LIN {X 0,Y 511.669,Z 782.628,A -85,B 0,C 180,E1 5380.533,E2 5380.533} C_VEL
LIN {X 0,Y 510.869,Z 808.748,A -85,B 0,C 180,E1 5382.068,E2 5382.068} C_VEL
LIN {X 0,Y 510.028,Z 830.874,A -85,B 0,C 180,E1 5384.067,E2 5384.067} C_VEL
LIN {X 0,Y 509.144,Z 850.479,A -85,B 0,C 180,E1 5386.68,E2 5386.68} C_VEL
LIN {X 0,Y 508.438,Z 865.261,A -85,B 0,C 180,E1 5389.712,E2 5389.712} C_VEL
LIN {X 0,Y 508.186,Z 873.103,A -85,B 0,C 180,E1 5392.299,E2 5392.299} C_VEL
LIN {X 0,Y 508.018,Z 877.24,A -85,B 0,C 180,E1 5394.874,E2 5394.874} C_VEL
LIN {X 0,Y 507.893,Z 877.639,A -85,B 0,C 180,E1 5398.296,E2 5398.296} C_VEL
LIN {X 0,Y 507.989,Z 872.219,A -85,B 0,C 180,E1 5401.712,E2 5401.712} C_VEL
LIN {X 0,Y 508.373,Z 861.446,A -85,B 0,C 180,E1 5404.859,E2 5404.859} C_VEL
LIN {X 0,Y 508.955,Z 845.862,A -85,B 0,C 180,E1 5407.697,E2 5407.697} C_VEL
LIN {X 0,Y 509.838,Z 824.739,A -85,B 0,C 180,E1 5410.267,E2 5410.267} C_VEL
LIN {X 0,Y 510.798,Z 799.503,A -85,B 0,C 180,E1 5412.304,E2 5412.304} C_VEL
LIN {X 0,Y 511.521,Z 770.953,A -85,B 0,C 180,E1 5413.749,E2 5413.749} C_VEL
LIN {X 0,Y 511.182,Z 749.928,A -85,B 0,C 180,E1 5414.374,E2 5414.374} C_VEL
LIN {X 0,Y 506.857,Z 733.66,A -85,B 0,C 180,E1 5414.896,E2 5414.896} C_VEL
LIN {X 0,Y 506.737,Z 733.66,A -85,B 0,C 180,E1 5421.014,E2 5421.014} C_VEL
LIN {X 0,Y 506.595,Z 733.66,A -85,B 0,C 180,E1 5426.638,E2 5426.638} C_VEL
LIN {X 0,Y 506.48,Z 733.66,A -85,B 0,C 180,E1 5432.557,E2 5432.557} C_VEL
LIN {X 0,Y 506.475,Z 733.66,A -85,B 0,C 180,E1 5436.722,E2 5436.722} C_VEL
LIN {X 0,Y 506.449,Z 733.66,A -85,B 0,C 180,E1 5443.444,E2 5443.444} C_VEL
LIN {X 0,Y 506.496,Z 733.66,A -85,B 0,C 180,E1 5448.879,E2 5448.879} C_VEL
LIN {X 0,Y 506.475,Z 733.66,A -85,B 0,C 180,E1 5455.389,E2 5455.389} C_VEL
LIN {X 0,Y 506.581,Z 733.66,A -85,B 0,C 180,E1 5459.288,E2 5459.288} C_VEL
LIN {X 0,Y 518.791,Z 764.917,A -85,B 0,C 180,E1 5460.693,E2 5460.693} C_VEL
LIN {X 0,Y 517.444,Z 800.699,A -85,B 0,C 180,E1 5461.845,E2 5461.845} C_VEL
LIN {X 0,Y 515.51,Z 834.822,A -85,B 0,C 180,E1 5463.6,E2 5463.6} C_VEL
LIN {X 0,Y 513.145,Z 867.936,A -85,B 0,C 180,E1 5466.042,E2 5466.042} C_VEL
LIN {X 0,Y 511.108,Z 896.809,A -85,B 0,C 180,E1 5468.952,E2 5468.952} C_VEL
LIN {X 0,Y 509.415,Z 921.908,A -85,B 0,C 180,E1 5472.332,E2 5472.332} C_VEL
LIN {X 0,Y 508.359,Z 943.041,A -85,B 0,C 180,E1 5476.216,E2 5476.216} C_VEL
LIN {X 0,Y 507.733,Z 958.105,A -85,B 0,C 180,E1 5480.168,E2 5480.168} C_VEL
LIN {X 0,Y 507.452,Z 967.534,A -85,B 0,C 180,E1 5484.006,E2 5484.006} C_VEL
LIN {X 0,Y 507.366,Z 972.536,A -85,B 0,C 180,E1 5488.29,E2 5488.29} C_VEL
LIN {X 0,Y 507.403,Z 972.482,A -85,B 0,C 180,E1 5491.71,E2 5491.71} C_VEL
LIN {X 0,Y 507.433,Z 967.371,A -85,B 0,C 180,E1 5495.995,E2 5495.995} C_VEL
LIN {X 0,Y 507.679,Z 957.879,A -85,B 0,C 180,E1 5499.818,E2 5499.818} C_VEL
LIN {X 0,Y 508.353,Z 941.596,A -85,B 0,C 180,E1 5504.012,E2 5504.012} C_VEL
LIN {X 0,Y 509.541,Z 919.84,A -85,B 0,C 180,E1 5507.894,E2 5507.894} C_VEL
LIN {X 0,Y 511.324,Z 894.013,A -85,B 0,C 180,E1 5511.284,E2 5511.284} C_VEL
LIN {X 0,Y 513.496,Z 862.942,A -85,B 0,C 180,E1 5514.286,E2 5514.286} C_VEL
LIN {X 0,Y 515.742,Z 829.441,A -85,B 0,C 180,E1 5516.641,E2 5516.641} C_VEL
LIN {X 0,Y 517.823,Z 792.141,A -85,B 0,C 180,E1 5518.403,E2 5518.403} C_VEL
LIN {X 0,Y 518.569,Z 762.784,A -85,B 0,C 180,E1 5519.287,E2 5519.287} C_VEL
LIN {X 0,Y 506.616,Z 733.66,A -85,B 0,C 180,E1 5520.704,E2 5520.704} C_VEL
LIN {X 0,Y 506.475,Z 733.66,A -85,B 0,C 180,E1 5526.72,E2 5526.72} C_VEL
LIN {X 0,Y 506.366,Z 733.66,A -85,B 0,C 180,E1 5533.451,E2 5533.451} C_VEL
LIN {X 0,Y 506.445,Z 733.66,A -85,B 0,C 180,E1 5538.871,E2 5538.871} C_VEL
LIN {X 0,Y 506.462,Z 733.66,A -85,B 0,C 180,E1 5545.386,E2 5545.386} C_VEL
LIN {X 0,Y 506.547,Z 733.66,A -85,B 0,C 180,E1 5551.426,E2 5551.426} C_VEL
LIN {X 0,Y 506.779,Z 733.66,A -85,B 0,C 180,E1 5557.848,E2 5557.848} C_VEL
LIN {X 0,Y 506.874,Z 733.66,A -85,B 0,C 180,E1 5562.917,E2 5562.917} C_VEL
LIN {X 0,Y 506.882,Z 733.66,A -85,B 0,C 180,E1 5569.672,E2 5569.672} C_VEL
LIN {X 0,Y 507.078,Z 733.66,A -85,B 0,C 180,E1 5574.857,E2 5574.857} C_VEL
LIN {X 0,Y 507.168,Z 733.66,A -85,B 0,C 180,E1 5579.996,E2 5579.996} C_VEL
LIN {X 0,Y 507.051,Z 733.66,A -85,B 0,C 180,E1 5585.135,E2 5585.135} C_VEL
LIN {X 0,Y 507.009,Z 733.66,A -85,B 0,C 180,E1 5590.317,E2 5590.317} C_VEL
LIN {X 0,Y 506.858,Z 733.66,A -85,B 0,C 180,E1 5595.591,E2 5595.591} C_VEL
LIN {X 0,Y 506.748,Z 733.66,A -85,B 0,C 180,E1 5601.005,E2 5601.005} C_VEL
LIN {X 0,Y 506.616,Z 733.66,A -85,B 0,C 180,E1 5606.629,E2 5606.629} C_VEL
LIN {X 0,Y 506.495,Z 733.66,A -85,B 0,C 180,E1 5612.547,E2 5612.547} C_VEL
LIN {X 0,Y 506.454,Z 733.66,A -85,B 0,C 180,E1 5616.714,E2 5616.714} C_VEL
LIN {X 0,Y 506.313,Z 733.66,A -85,B 0,C 180,E1 5620.319,E2 5620.319} C_VEL
LIN {X 0,Y 503.847,Z 733.66,A -85,B 0,C 180,E1 5621.78,E2 5621.78} C_VEL
LIN {X 0,Y 498.62,Z 733.66,A -85,B 0,C 180,E1 5623.971,E2 5623.971} C_VEL
LIN {X 0,Y 498.547,Z 733.66,A -85,B 0,C 180,E1 5624.224,E2 5624.224} C_VEL
LIN {X 0,Y 498.53,Z 733.66,A -85,B 0,C 180,E1 5630.372,E2 5630.372} C_VEL
LIN {X 0,Y 498.636,Z 734.246,A -85,B 0,C 180,E1 5636.385,E2 5636.385} C_VEL
LIN {X 0,Y 507.42,Z 762.538,A -85,B 0,C 180,E1 5638.882,E2 5638.882} C_VEL
LIN {X 0,Y 512.218,Z 771.17,A -85,B 0,C 180,E1 5639.711,E2 5639.711} C_VEL
LIN {X 0,Y 511.027,Z 821.133,A -85,B 0,C 180,E1 5640.64,E2 5640.64} C_VEL
LIN {X 0,Y 509.28,Z 859.027,A -85,B 0,C 180,E1 5642.019,E2 5642.019} C_VEL
LIN {X 0,Y 507.142,Z 895.986,A -85,B 0,C 180,E1 5644.11,E2 5644.11} C_VEL
LIN {X 0,Y 504.962,Z 929.253,A -85,B 0,C 180,E1 5646.777,E2 5646.777} C_VEL
LIN {X 0,Y 502.727,Z 958.925,A -85,B 0,C 180,E1 5650.195,E2 5650.195} C_VEL
LIN {X 0,Y 501.04,Z 982.915,A -85,B 0,C 180,E1 5653.993,E2 5653.993} C_VEL
LIN {X 0,Y 500.101,Z 1000.207,A -85,B 0,C 180,E1 5657.764,E2 5657.764} C_VEL
LIN {X 0,Y 499.71,Z 1012.766,A -85,B 0,C 180,E1 5661.725,E2 5661.725} C_VEL
LIN {X 0,Y 499.517,Z 1020.156,A -85,B 0,C 180,E1 5665.654,E2 5665.654} C_VEL
LIN {X 0,Y 499.462,Z 1023,A -85,B 0,C 180,E1 5670,E2 5670} C_VEL
LIN {X 0,Y 499.572,Z 1020.161,A -85,B 0,C 180,E1 5674.345,E2 5674.345} C_VEL
LIN {X 0,Y 499.739,Z 1011.589,A -85,B 0,C 180,E1 5678.713,E2 5678.713} C_VEL
LIN {X 0,Y 500.185,Z 998.527,A -85,B 0,C 180,E1 5682.677,E2 5682.677} C_VEL
LIN {X 0,Y 501.216,Z 979.219,A -85,B 0,C 180,E1 5686.677,E2 5686.677} C_VEL
LIN {X 0,Y 502.895,Z 955.449,A -85,B 0,C 180,E1 5690.257,E2 5690.257} C_VEL
LIN {X 0,Y 505.025,Z 927.806,A -85,B 0,C 180,E1 5693.359,E2 5693.359} C_VEL
LIN {X 0,Y 507.005,Z 896.867,A -85,B 0,C 180,E1 5695.778,E2 5695.778} C_VEL
LIN {X 0,Y 508.885,Z 859.818,A -85,B 0,C 180,E1 5697.823,E2 5697.823} C_VEL
LIN {X 0,Y 510.524,Z 822.877,A -85,B 0,C 180,E1 5699.209,E2 5699.209} C_VEL
LIN {X 0,Y 511.5,Z 775.815,A -85,B 0,C 180,E1 5700.099,E2 5700.099} C_VEL
LIN {X 0,Y 511.122,Z 768.237,A -85,B 0,C 180,E1 5700.244,E2 5700.244} C_VEL
LIN {X 0,Y 502.858,Z 752.585,A -85,B 0,C 180,E1 5701.5,E2 5701.5} C_VEL
LIN {X 0,Y 498.702,Z 733.66,A -85,B 0,C 180,E1 5702.958,E2 5702.958} C_VEL
LIN {X 0,Y 498.518,Z 733.66,A -85,B 0,C 180,E1 5709.628,E2 5709.628} C_VEL
LIN {X 0,Y 498.549,Z 733.66,A -85,B 0,C 180,E1 5715.701,E2 5715.701} C_VEL
LIN {X 0,Y 498.458,Z 733.66,A -85,B 0,C 180,E1 5722.163,E2 5722.163} C_VEL
LIN {X 0,Y 498.613,Z 733.66,A -85,B 0,C 180,E1 5728.239,E2 5728.239} C_VEL
LIN {X 0,Y 498.667,Z 733.66,A -85,B 0,C 180,E1 5734.85,E2 5734.85} C_VEL
LIN {X 0,Y 498.822,Z 733.836,A -85,B 0,C 180,E1 5738.675,E2 5738.675} C_VEL
LIN {X 0,Y 504.418,Z 756.647,A -85,B 0,C 180,E1 5739.358,E2 5739.358} C_VEL
LIN {X 0,Y 504.167,Z 784.832,A -85,B 0,C 180,E1 5740.315,E2 5740.315} C_VEL
LIN {X 0,Y 503.319,Z 811.126,A -85,B 0,C 180,E1 5741.915,E2 5741.915} C_VEL
LIN {X 0,Y 502.421,Z 833.815,A -85,B 0,C 180,E1 5744.044,E2 5744.044} C_VEL
LIN {X 0,Y 501.469,Z 852.859,A -85,B 0,C 180,E1 5746.695,E2 5746.695} C_VEL
LIN {X 0,Y 500.743,Z 866.419,A -85,B 0,C 180,E1 5749.552,E2 5749.552} C_VEL
LIN {X 0,Y 500.412,Z 874.294,A -85,B 0,C 180,E1 5752.179,E2 5752.179} C_VEL
LIN {X 0,Y 500.245,Z 878.482,A -85,B 0,C 180,E1 5754.795,E2 5754.795} C_VEL
LIN {X 0,Y 500.101,Z 878.894,A -85,B 0,C 180,E1 5758.269,E2 5758.269} C_VEL
LIN {X 0,Y 500.209,Z 873.502,A -85,B 0,C 180,E1 5761.738,E2 5761.738} C_VEL
LIN {X 0,Y 500.615,Z 863.453,A -85,B 0,C 180,E1 5764.775,E2 5764.775} C_VEL
LIN {X 0,Y 501.268,Z 847.192,A -85,B 0,C 180,E1 5767.816,E2 5767.816} C_VEL
LIN {X 0,Y 502.208,Z 826.16,A -85,B 0,C 180,E1 5770.425,E2 5770.425} C_VEL
LIN {X 0,Y 503.228,Z 801.1,A -85,B 0,C 180,E1 5772.492,E2 5772.492} C_VEL
LIN {X 0,Y 504.04,Z 772.436,A -85,B 0,C 180,E1 5773.979,E2 5773.979} C_VEL
LIN {X 0,Y 503.662,Z 751.113,A -85,B 0,C 180,E1 5774.633,E2 5774.633} C_VEL
LIN {X 0,Y 498.945,Z 733.66,A -85,B 0,C 180,E1 5775.202,E2 5775.202} C_VEL
LIN {X 0,Y 498.833,Z 733.66,A -85,B 0,C 180,E1 5781.363,E2 5781.363} C_VEL
LIN {X 0,Y 498.622,Z 733.66,A -85,B 0,C 180,E1 5787.099,E2 5787.099} C_VEL
LIN {X 0,Y 498.57,Z 733.66,A -85,B 0,C 180,E1 5793.139,E2 5793.139} C_VEL
LIN {X 0,Y 498.438,Z 733.66,A -85,B 0,C 180,E1 5799.639,E2 5799.639} C_VEL
LIN {X 0,Y 498.578,Z 733.66,A -85,B 0,C 180,E1 5805.696,E2 5805.696} C_VEL
LIN {X 0,Y 498.515,Z 733.66,A -85,B 0,C 180,E1 5812.157,E2 5812.157} C_VEL
LIN {X 0,Y 498.667,Z 733.66,A -85,B 0,C 180,E1 5818.734,E2 5818.734} C_VEL
LIN {X 0,Y 511.844,Z 767.711,A -85,B 0,C 180,E1 5820.322,E2 5820.322} C_VEL
LIN {X 0,Y 510.29,Z 804.648,A -85,B 0,C 180,E1 5821.577,E2 5821.577} C_VEL
LIN {X 0,Y 508.123,Z 839.115,A -85,B 0,C 180,E1 5823.451,E2 5823.451} C_VEL
LIN {X 0,Y 505.598,Z 870.976,A -85,B 0,C 180,E1 5825.928,E2 5825.928} C_VEL
LIN {X 0,Y 503.261,Z 901.087,A -85,B 0,C 180,E1 5829.132,E2 5829.132} C_VEL
LIN {X 0,Y 501.474,Z 925.585,A -85,B 0,C 180,E1 5832.653,E2 5832.653} C_VEL
LIN {X 0,Y 500.419,Z 944.967,A -85,B 0,C 180,E1 5836.439,E2 5836.439} C_VEL
LIN {X 0,Y 499.823,Z 959.67,A -85,B 0,C 180,E1 5840.531,E2 5840.531} C_VEL
LIN {X 0,Y 499.512,Z 969.032,A -85,B 0,C 180,E1 5844.783,E2 5844.783} C_VEL
LIN {X 0,Y 499.465,Z 972.536,A -85,B 0,C 180,E1 5848.263,E2 5848.263} C_VEL
LIN {X 0,Y 499.524,Z 972.482,A -85,B 0,C 180,E1 5851.737,E2 5851.737} C_VEL
LIN {X 0,Y 499.548,Z 967.373,A -85,B 0,C 180,E1 5856.09,E2 5856.09} C_VEL
LIN {X 0,Y 499.837,Z 957.218,A -85,B 0,C 180,E1 5860.194,E2 5860.194} C_VEL
LIN {X 0,Y 500.609,Z 940.668,A -85,B 0,C 180,E1 5864.427,E2 5864.427} C_VEL
LIN {X 0,Y 501.862,Z 919.842,A -85,B 0,C 180,E1 5868.177,E2 5868.177} C_VEL
LIN {X 0,Y 503.825,Z 894.152,A -85,B 0,C 180,E1 5871.6,E2 5871.6} C_VEL
LIN {X 0,Y 506.216,Z 863.768,A -85,B 0,C 180,E1 5874.615,E2 5874.615} C_VEL
LIN {X 0,Y 508.625,Z 830.535,A -85,B 0,C 180,E1 5876.998,E2 5876.998} C_VEL
LIN {X 0,Y 510.844,Z 793.534,A -85,B 0,C 180,E1 5878.788,E2 5878.788} C_VEL
LIN {X 0,Y 511.555,Z 764.744,A -85,B 0,C 180,E1 5879.685,E2 5879.685} C_VEL
LIN {X 0,Y 498.703,Z 733.66,A -85,B 0,C 180,E1 5881.245,E2 5881.245} C_VEL
LIN {X 0,Y 498.472,Z 733.66,A -85,B 0,C 180,E1 5887.409,E2 5887.409} C_VEL
LIN {X 0,Y 498.436,Z 733.66,A -85,B 0,C 180,E1 5893.191,E2 5893.191} C_VEL
LIN {X 0,Y 498.479,Z 733.66,A -85,B 0,C 180,E1 5899.408,E2 5899.408} C_VEL
LIN {X 0,Y 498.554,Z 733.66,A -85,B 0,C 180,E1 5905.083,E2 5905.083} C_VEL
LIN {X 0,Y 498.627,Z 733.66,A -85,B 0,C 180,E1 5911.715,E2 5911.715} C_VEL
LIN {X 0,Y 498.805,Z 733.66,A -85,B 0,C 180,E1 5916.756,E2 5916.756} C_VEL
LIN {X 0,Y 498.928,Z 733.66,A -85,B 0,C 180,E1 5922.331,E2 5922.331} C_VEL
LIN {X 0,Y 498.818,Z 733.66,A -85,B 0,C 180,E1 5927.729,E2 5927.729} C_VEL
LIN {X 0,Y 499.173,Z 733.66,A -85,B 0,C 180,E1 5933.028,E2 5933.028} C_VEL
LIN {X 0,Y 499.419,Z 733.66,A -85,B 0,C 180,E1 5938.259,E2 5938.259} C_VEL
LIN {X 0,Y 499.308,Z 733.66,A -85,B 0,C 180,E1 5943.473,E2 5943.473} C_VEL
LIN {X 0,Y 499.122,Z 733.66,A -85,B 0,C 180,E1 5948.72,E2 5948.72} C_VEL
LIN {X 0,Y 498.986,Z 733.66,A -85,B 0,C 180,E1 5954.044,E2 5954.044} C_VEL
LIN {X 0,Y 498.859,Z 733.66,A -85,B 0,C 180,E1 5959.799,E2 5959.799} C_VEL
LIN {X 0,Y 498.742,Z 733.66,A -85,B 0,C 180,E1 5965.146,E2 5965.146} C_VEL
LIN {X 0,Y 498.567,Z 733.66,A -85,B 0,C 180,E1 5971.752,E2 5971.752} C_VEL
LIN {X 0,Y 498.446,Z 733.66,A -85,B 0,C 180,E1 5977.834,E2 5977.834} C_VEL
LIN {X 0,Y 498.547,Z 733.66,A -85,B 0,C 180,E1 5984.224,E2 5984.224} C_VEL
LIN {X 0,Y 496.117,Z 733.66,A -85,B 0,C 180,E1 5985.7,E2 5985.7} C_VEL
LIN {X 0,Y 490.625,Z 733.66,A -85,B 0,C 180,E1 5988.168,E2 5988.168} C_VEL
LIN {X 0,Y 490.589,Z 733.66,A -85,B 0,C 180,E1 5994.098,E2 5994.098} C_VEL
LIN {X 0,Y 490.728,Z 734.334,A -85,B 0,C 180,E1 5995.891,E2 5995.891} C_VEL
LIN {X 0,Y 500.518,Z 766.213,A -85,B 0,C 180,E1 5998.771,E2 5998.771} C_VEL
LIN {X 0,Y 505.014,Z 773.789,A -85,B 0,C 180,E1 5999.357,E2 5999.357} C_VEL
LIN {X 0,Y 503.827,Z 821.165,A -85,B 0,C 180,E1 6000.266,E2 6000.266} C_VEL
LIN {X 0,Y 501.909,Z 859.192,A -85,B 0,C 180,E1 6001.694,E2 6001.694} C_VEL
LIN {X 0,Y 499.659,Z 895.278,A -85,B 0,C 180,E1 6003.778,E2 6003.778} C_VEL
LIN {X 0,Y 497.339,Z 928.358,A -85,B 0,C 180,E1 6006.464,E2 6006.464} C_VEL
LIN {X 0,Y 495.236,Z 957.423,A -85,B 0,C 180,E1 6009.688,E2 6009.688} C_VEL
LIN {X 0,Y 493.435,Z 980.441,A -85,B 0,C 180,E1 6013.281,E2 6013.281} C_VEL
LIN {X 0,Y 492.398,Z 998.525,A -85,B 0,C 180,E1 6017.118,E2 6017.118} C_VEL
LIN {X 0,Y 491.832,Z 1012.767,A -85,B 0,C 180,E1 6021.591,E2 6021.591} C_VEL
LIN {X 0,Y 491.634,Z 1020.151,A -85,B 0,C 180,E1 6025.584,E2 6025.584} C_VEL
LIN {X 0,Y 491.562,Z 1023,A -85,B 0,C 180,E1 6030,E2 6030} C_VEL
LIN {X 0,Y 491.686,Z 1020.156,A -85,B 0,C 180,E1 6034.415,E2 6034.415} C_VEL
LIN {X 0,Y 491.849,Z 1011.585,A -85,B 0,C 180,E1 6038.854,E2 6038.854} C_VEL
LIN {X 0,Y 492.361,Z 998.531,A -85,B 0,C 180,E1 6042.882,E2 6042.882} C_VEL
LIN {X 0,Y 493.457,Z 979.215,A -85,B 0,C 180,E1 6046.947,E2 6046.947} C_VEL
LIN {X 0,Y 495.183,Z 957.421,A -85,B 0,C 180,E1 6050.313,E2 6050.313} C_VEL
LIN {X 0,Y 497.144,Z 929.961,A -85,B 0,C 180,E1 6053.323,E2 6053.323} C_VEL
LIN {X 0,Y 499.641,Z 893.617,A -85,B 0,C 180,E1 6056.23,E2 6056.23} C_VEL
LIN {X 0,Y 501.836,Z 859.318,A -85,B 0,C 180,E1 6058.249,E2 6058.249} C_VEL
LIN {X 0,Y 503.544,Z 823.942,A -85,B 0,C 180,E1 6059.609,E2 6059.609} C_VEL
LIN {X 0,Y 504.605,Z 780.158,A -85,B 0,C 180,E1 6060.481,E2 6060.481} C_VEL
LIN {X 0,Y 504.079,Z 771.093,A -85,B 0,C 180,E1 6060.662,E2 6060.662} C_VEL
LIN {X 0,Y 496.028,Z 756.848,A -85,B 0,C 180,E1 6061.482,E2 6061.482} C_VEL
LIN {X 0,Y 490.79,Z 733.66,A -85,B 0,C 180,E1 6063.259,E2 6063.259} C_VEL
LIN {X 0,Y 490.603,Z 733.66,A -85,B 0,C 180,E1 6069.517,E2 6069.517} C_VEL
LIN {X 0,Y 490.631,Z 733.66,A -85,B 0,C 180,E1 6075.217,E2 6075.217} C_VEL
LIN {X 0,Y 490.53,Z 733.66,A -85,B 0,C 180,E1 6080.503,E2 6080.503} C_VEL
LIN {X 0,Y 490.695,Z 733.66,A -85,B 0,C 180,E1 6086.42,E2 6086.42} C_VEL
LIN {X 0,Y 490.662,Z 733.66,A -85,B 0,C 180,E1 6092.434,E2 6092.434} C_VEL
LIN {X 0,Y 490.838,Z 733.66,A -85,B 0,C 180,E1 6098.28,E2 6098.28} C_VEL
LIN {X 0,Y 497.028,Z 758.522,A -85,B 0,C 180,E1 6099.088,E2 6099.088} C_VEL
LIN {X 0,Y 496.702,Z 787.762,A -85,B 0,C 180,E1 6100.123,E2 6100.123} C_VEL
LIN {X 0,Y 495.784,Z 813.888,A -85,B 0,C 180,E1 6101.778,E2 6101.778} C_VEL
LIN {X 0,Y 494.749,Z 836.769,A -85,B 0,C 180,E1 6104.017,E2 6104.017} C_VEL
LIN {X 0,Y 493.748,Z 855.208,A -85,B 0,C 180,E1 6106.708,E2 6106.708} C_VEL
LIN {X 0,Y 492.908,Z 869.633,A -85,B 0,C 180,E1 6109.951,E2 6109.951} C_VEL
LIN {X 0,Y 492.586,Z 877.302,A -85,B 0,C 180,E1 6112.942,E2 6112.942} C_VEL
LIN {X 0,Y 492.309,Z 880.672,A -85,B 0,C 180,E1 6116.478,E2 6116.478} C_VEL
LIN {X 0,Y 492.342,Z 878.211,A -85,B 0,C 180,E1 6120.004,E2 6120.004} C_VEL
LIN {X 0,Y 492.617,Z 870.978,A -85,B 0,C 180,E1 6123.131,E2 6123.131} C_VEL
LIN {X 0,Y 493.184,Z 857.531,A -85,B 0,C 180,E1 6126.393,E2 6126.393} C_VEL
LIN {X 0,Y 494.007,Z 839.068,A -85,B 0,C 180,E1 6129.263,E2 6129.263} C_VEL
LIN {X 0,Y 495.028,Z 816.427,A -85,B 0,C 180,E1 6131.639,E2 6131.639} C_VEL
LIN {X 0,Y 496.106,Z 789.979,A -85,B 0,C 180,E1 6133.46,E2 6133.46} C_VEL
LIN {X 0,Y 496.818,Z 760.529,A -85,B 0,C 180,E1 6134.662,E2 6134.662} C_VEL
LIN {X 0,Y 494.672,Z 747.189,A -85,B 0,C 180,E1 6135.054,E2 6135.054} C_VEL
LIN {X 0,Y 490.995,Z 733.66,A -85,B 0,C 180,E1 6135.54,E2 6135.54} C_VEL
LIN {X 0,Y 490.878,Z 733.66,A -85,B 0,C 180,E1 6141.727,E2 6141.727} C_VEL
LIN {X 0,Y 490.682,Z 733.66,A -85,B 0,C 180,E1 6147.574,E2 6147.574} C_VEL
LIN {X 0,Y 490.635,Z 733.66,A -85,B 0,C 180,E1 6153.746,E2 6153.746} C_VEL
LIN {X 0,Y 490.521,Z 733.66,A -85,B 0,C 180,E1 6160.409,E2 6160.409} C_VEL
LIN {X 0,Y 490.651,Z 733.66,A -85,B 0,C 180,E1 6165.217,E2 6165.217} C_VEL
LIN {X 0,Y 490.609,Z 733.66,A -85,B 0,C 180,E1 6170.494,E2 6170.494} C_VEL
LIN {X 0,Y 490.6,Z 733.66,A -85,B 0,C 180,E1 6176.439,E2 6176.439} C_VEL
LIN {X 0,Y 490.7,Z 734.051,A -85,B 0,C 180,E1 6178.209,E2 6178.209} C_VEL
LIN {X 0,Y 504.974,Z 769.857,A -85,B 0,C 180,E1 6179.928,E2 6179.928} C_VEL
LIN {X 0,Y 503.168,Z 807.933,A -85,B 0,C 180,E1 6181.281,E2 6181.281} C_VEL
LIN {X 0,Y 500.738,Z 842.932,A -85,B 0,C 180,E1 6183.281,E2 6183.281} C_VEL
LIN {X 0,Y 498.092,Z 874.664,A -85,B 0,C 180,E1 6185.863,E2 6185.863} C_VEL
LIN {X 0,Y 495.572,Z 903.255,A -85,B 0,C 180,E1 6189.059,E2 6189.059} C_VEL
LIN {X 0,Y 493.62,Z 928.201,A -85,B 0,C 180,E1 6192.829,E2 6192.829} C_VEL
LIN {X 0,Y 492.507,Z 946.89,A -85,B 0,C 180,E1 6196.67,E2 6196.67} C_VEL
LIN {X 0,Y 491.931,Z 960.249,A -85,B 0,C 180,E1 6200.576,E2 6200.576} C_VEL
LIN {X 0,Y 491.614,Z 969.031,A -85,B 0,C 180,E1 6204.699,E2 6204.699} C_VEL
LIN {X 0,Y 491.563,Z 972.535,A -85,B 0,C 180,E1 6208.235,E2 6208.235} C_VEL
LIN {X 0,Y 491.621,Z 972.482,A -85,B 0,C 180,E1 6211.765,E2 6211.765} C_VEL
LIN {X 0,Y 491.674,Z 967.374,A -85,B 0,C 180,E1 6216.188,E2 6216.188} C_VEL
LIN {X 0,Y 491.951,Z 957.683,A -85,B 0,C 180,E1 6220.203,E2 6220.203} C_VEL
LIN {X 0,Y 492.792,Z 941.299,A -85,B 0,C 180,E1 6224.527,E2 6224.527} C_VEL
LIN {X 0,Y 494.194,Z 920.07,A -85,B 0,C 180,E1 6228.433,E2 6228.433} C_VEL
LIN {X 0,Y 496.39,Z 894.463,A -85,B 0,C 180,E1 6231.941,E2 6231.941} C_VEL
LIN {X 0,Y 498.991,Z 864.175,A -85,B 0,C 180,E1 6234.995,E2 6234.995} C_VEL
LIN {X 0,Y 501.564,Z 830.905,A -85,B 0,C 180,E1 6237.411,E2 6237.411} C_VEL
LIN {X 0,Y 503.905,Z 794.756,A -85,B 0,C 180,E1 6239.188,E2 6239.188} C_VEL
LIN {X 0,Y 504.444,Z 766.667,A -85,B 0,C 180,E1 6240.103,E2 6240.103} C_VEL
LIN {X 0,Y 490.758,Z 733.66,A -85,B 0,C 180,E1 6241.791,E2 6241.791} C_VEL
LIN {X 0,Y 490.53,Z 733.66,A -85,B 0,C 180,E1 6248.122,E2 6248.122} C_VEL
LIN {X 0,Y 490.596,Z 733.66,A -85,B 0,C 180,E1 6254.776,E2 6254.776} C_VEL
LIN {X 0,Y 490.57,Z 733.66,A -85,B 0,C 180,E1 6260.498,E2 6260.498} C_VEL
LIN {X 0,Y 490.592,Z 733.66,A -85,B 0,C 180,E1 6266.439,E2 6266.439} C_VEL
LIN {X 0,Y 490.73,Z 733.66,A -85,B 0,C 180,E1 6272.429,E2 6272.429} C_VEL
LIN {X 0,Y 490.933,Z 733.66,A -85,B 0,C 180,E1 6278.276,E2 6278.276} C_VEL
LIN {X 0,Y 490.924,Z 733.66,A -85,B 0,C 180,E1 6283.881,E2 6283.881} C_VEL
LIN {X 0,Y 491.047,Z 733.66,A -85,B 0,C 180,E1 6290.642,E2 6290.642} C_VEL
LIN {X 0,Y 491.225,Z 733.66,A -85,B 0,C 180,E1 6296.462,E2 6296.462} C_VEL
LIN {X 0,Y 491.289,Z 733.66,A -85,B 0,C 180,E1 6301.762,E2 6301.762} C_VEL
LIN {X 0,Y 491.155,Z 733.66,A -85,B 0,C 180,E1 6307.079,E2 6307.079} C_VEL
LIN {X 0,Y 491.063,Z 733.66,A -85,B 0,C 180,E1 6312.459,E2 6312.459} C_VEL
LIN {X 0,Y 490.978,Z 733.66,A -85,B 0,C 180,E1 6317.957,E2 6317.957} C_VEL
LIN {X 0,Y 490.838,Z 733.66,A -85,B 0,C 180,E1 6323.636,E2 6323.636} C_VEL
LIN {X 0,Y 490.641,Z 733.66,A -85,B 0,C 180,E1 6330.223,E2 6330.223} C_VEL
LIN {X 0,Y 490.543,Z 733.66,A -85,B 0,C 180,E1 6335.898,E2 6335.898} C_VEL
LIN {X 0,Y 490.618,Z 733.66,A -85,B 0,C 180,E1 6342.212,E2 6342.212} C_VEL
LIN {X 0,Y 490.625,Z 733.66,A -85,B 0,C 180,E1 6348.168,E2 6348.168} C_VEL
LIN {X 0,Y 486.608,Z 733.66,A -85,B 0,C 180,E1 6350.151,E2 6350.151} C_VEL
LIN {X 0,Y 482.63,Z 733.66,A -85,B 0,C 180,E1 6352.165,E2 6352.165} C_VEL
LIN {X 0,Y 482.809,Z 734.18,A -85,B 0,C 180,E1 6355.386,E2 6355.386} C_VEL
LIN {X 0,Y 493.608,Z 769.811,A -85,B 0,C 180,E1 6358.597,E2 6358.597} C_VEL
LIN {X 0,Y 497.682,Z 775.9,A -85,B 0,C 180,E1 6358.959,E2 6358.959} C_VEL
LIN {X 0,Y 496.678,Z 822.788,A -85,B 0,C 180,E1 6359.913,E2 6359.913} C_VEL
LIN {X 0,Y 494.694,Z 858.971,A -85,B 0,C 180,E1 6361.305,E2 6361.305} C_VEL
LIN {X 0,Y 492.066,Z 896.173,A -85,B 0,C 180,E1 6363.547,E2 6363.547} C_VEL
LIN {X 0,Y 489.624,Z 928.895,A -85,B 0,C 180,E1 6366.296,E2 6366.296} C_VEL
LIN {X 0,Y 487.393,Z 958.43,A -85,B 0,C 180,E1 6369.649,E2 6369.649} C_VEL
LIN {X 0,Y 485.639,Z 981.652,A -85,B 0,C 180,E1 6373.238,E2 6373.238} C_VEL
LIN {X 0,Y 484.457,Z 1000.196,A -85,B 0,C 180,E1 6377.363,E2 6377.363} C_VEL
LIN {X 0,Y 483.958,Z 1012.766,A -85,B 0,C 180,E1 6381.454,E2 6381.454} C_VEL
LIN {X 0,Y 483.749,Z 1020.146,A -85,B 0,C 180,E1 6385.512,E2 6385.512} C_VEL
LIN {X 0,Y 483.67,Z 1023,A -85,B 0,C 180,E1 6390,E2 6390} C_VEL
LIN {X 0,Y 483.795,Z 1020.152,A -85,B 0,C 180,E1 6394.487,E2 6394.487} C_VEL
LIN {X 0,Y 483.977,Z 1011.582,A -85,B 0,C 180,E1 6398.999,E2 6398.999} C_VEL
LIN {X 0,Y 484.56,Z 998.534,A -85,B 0,C 180,E1 6403.093,E2 6403.093} C_VEL
LIN {X 0,Y 485.762,Z 979.13,A -85,B 0,C 180,E1 6407.224,E2 6407.224} C_VEL
LIN {X 0,Y 487.366,Z 956.573,A -85,B 0,C 180,E1 6410.534,E2 6410.534} C_VEL
LIN {X 0,Y 490.078,Z 921.521,A -85,B 0,C 180,E1 6414.32,E2 6414.32} C_VEL
LIN {X 0,Y 492.645,Z 889.446,A -85,B 0,C 180,E1 6416.908,E2 6416.908} C_VEL
LIN {X 0,Y 495.052,Z 855.282,A -85,B 0,C 180,E1 6418.859,E2 6418.859} C_VEL
LIN {X 0,Y 496.961,Z 818.586,A -85,B 0,C 180,E1 6420.203,E2 6420.203} C_VEL
LIN {X 0,Y 497.338,Z 774.54,A -85,B 0,C 180,E1 6421.064,E2 6421.064} C_VEL
LIN {X 0,Y 488.141,Z 756.629,A -85,B 0,C 180,E1 6422.017,E2 6422.017} C_VEL
LIN {X 0,Y 485.394,Z 746.114,A -85,B 0,C 180,E1 6422.638,E2 6422.638} C_VEL
LIN {X 0,Y 482.828,Z 733.66,A -85,B 0,C 180,E1 6423.674,E2 6423.674} C_VEL
LIN {X 0,Y 482.658,Z 733.66,A -85,B 0,C 180,E1 6428.858,E2 6428.858} C_VEL
LIN {X 0,Y 482.679,Z 733.66,A -85,B 0,C 180,E1 6433.833,E2 6433.833} C_VEL
LIN {X 0,Y 482.612,Z 733.66,A -85,B 0,C 180,E1 6438.846,E2 6438.846} C_VEL
LIN {X 0,Y 482.679,Z 733.66,A -85,B 0,C 180,E1 6445.63,E2 6445.63} C_VEL
LIN {X 0,Y 482.705,Z 733.66,A -85,B 0,C 180,E1 6451.939,E2 6451.939} C_VEL
LIN {X 0,Y 482.89,Z 733.66,A -85,B 0,C 180,E1 6457.87,E2 6457.87} C_VEL
LIN {X 0,Y 489.616,Z 758.27,A -85,B 0,C 180,E1 6458.747,E2 6458.747} C_VEL
LIN {X 0,Y 489.371,Z 786.965,A -85,B 0,C 180,E1 6459.736,E2 6459.736} C_VEL
LIN {X 0,Y 488.428,Z 813.246,A -85,B 0,C 180,E1 6461.362,E2 6461.362} C_VEL
LIN {X 0,Y 487.352,Z 835.892,A -85,B 0,C 180,E1 6463.536,E2 6463.536} C_VEL
LIN {X 0,Y 486.226,Z 855.105,A -85,B 0,C 180,E1 6466.269,E2 6466.269} C_VEL
LIN {X 0,Y 485.37,Z 868.786,A -85,B 0,C 180,E1 6469.217,E2 6469.217} C_VEL
LIN {X 0,Y 484.893,Z 876.715,A -85,B 0,C 180,E1 6471.927,E2 6471.927} C_VEL
LIN {X 0,Y 484.716,Z 880.98,A -85,B 0,C 180,E1 6474.627,E2 6474.627} C_VEL
LIN {X 0,Y 484.525,Z 881.42,A -85,B 0,C 180,E1 6478.213,E2 6478.213} C_VEL
LIN {X 0,Y 484.655,Z 876.05,A -85,B 0,C 180,E1 6481.794,E2 6481.794} C_VEL
LIN {X 0,Y 485.121,Z 866.033,A -85,B 0,C 180,E1 6484.927,E2 6484.927} C_VEL
LIN {X 0,Y 485.87,Z 849.821,A -85,B 0,C 180,E1 6488.065,E2 6488.065} C_VEL
LIN {X 0,Y 486.923,Z 828.912,A -85,B 0,C 180,E1 6490.756,E2 6490.756} C_VEL
LIN {X 0,Y 488.077,Z 804.161,A -85,B 0,C 180,E1 6492.887,E2 6492.887} C_VEL
LIN {X 0,Y 488.993,Z 776.266,A -85,B 0,C 180,E1 6494.415,E2 6494.415} C_VEL
LIN {X 0,Y 488.701,Z 754.307,A -85,B 0,C 180,E1 6495.144,E2 6495.144} C_VEL
LIN {X 0,Y 483.07,Z 733.66,A -85,B 0,C 180,E1 6495.769,E2 6495.769} C_VEL
LIN {X 0,Y 482.957,Z 733.66,A -85,B 0,C 180,E1 6502.102,E2 6502.102} C_VEL
LIN {X 0,Y 482.68,Z 733.66,A -85,B 0,C 180,E1 6508.561,E2 6508.561} C_VEL
LIN {X 0,Y 482.641,Z 733.66,A -85,B 0,C 180,E1 6514.383,E2 6514.383} C_VEL
LIN {X 0,Y 482.605,Z 733.66,A -85,B 0,C 180,E1 6518.866,E2 6518.866} C_VEL
LIN {X 0,Y 482.649,Z 733.66,A -85,B 0,C 180,E1 6523.82,E2 6523.82} C_VEL
LIN {X 0,Y 482.695,Z 733.66,A -85,B 0,C 180,E1 6528.838,E2 6528.838} C_VEL
LIN {X 0,Y 482.623,Z 733.66,A -85,B 0,C 180,E1 6534.657,E2 6534.657} C_VEL
LIN {X 0,Y 482.727,Z 733.66,A -85,B 0,C 180,E1 6537.585,E2 6537.585} C_VEL
LIN {X 0,Y 498.097,Z 772.095,A -85,B 0,C 180,E1 6539.524,E2 6539.524} C_VEL
LIN {X 0,Y 496.151,Z 809.441,A -85,B 0,C 180,E1 6540.899,E2 6540.899} C_VEL
LIN {X 0,Y 493.595,Z 843.856,A -85,B 0,C 180,E1 6542.905,E2 6542.905} C_VEL
LIN {X 0,Y 490.696,Z 876.26,A -85,B 0,C 180,E1 6545.595,E2 6545.595} C_VEL
LIN {X 0,Y 488.017,Z 904.414,A -85,B 0,C 180,E1 6548.826,E2 6548.826} C_VEL
LIN {X 0,Y 485.926,Z 928.345,A -85,B 0,C 180,E1 6552.548,E2 6552.548} C_VEL
LIN {X 0,Y 484.575,Z 948.661,A -85,B 0,C 180,E1 6556.907,E2 6556.907} C_VEL
LIN {X 0,Y 483.96,Z 961.719,A -85,B 0,C 180,E1 6561.001,E2 6561.001} C_VEL
LIN {X 0,Y 483.693,Z 970.229,A -85,B 0,C 180,E1 6565.512,E2 6565.512} C_VEL
LIN {X 0,Y 483.716,Z 972.998,A -85,B 0,C 180,E1 6570,E2 6570} C_VEL
LIN {X 0,Y 483.784,Z 970.106,A -85,B 0,C 180,E1 6574.488,E2 6574.488} C_VEL
LIN {X 0,Y 483.953,Z 961.496,A -85,B 0,C 180,E1 6579,E2 6579} C_VEL
LIN {X 0,Y 484.52,Z 948.323,A -85,B 0,C 180,E1 6583.095,E2 6583.095} C_VEL
LIN {X 0,Y 485.934,Z 927.85,A -85,B 0,C 180,E1 6587.452,E2 6587.452} C_VEL
LIN {X 0,Y 487.958,Z 904.664,A -85,B 0,C 180,E1 6591.052,E2 6591.052} C_VEL
LIN {X 0,Y 490.592,Z 877.066,A -85,B 0,C 180,E1 6594.237,E2 6594.237} C_VEL
LIN {X 0,Y 493.499,Z 844.976,A -85,B 0,C 180,E1 6596.927,E2 6596.927} C_VEL
LIN {X 0,Y 496.148,Z 811.248,A -85,B 0,C 180,E1 6598.915,E2 6598.915} C_VEL
LIN {X 0,Y 498.008,Z 776.729,A -85,B 0,C 180,E1 6600.248,E2 6600.248} C_VEL
LIN {X 0,Y 497.176,Z 767.9,A -85,B 0,C 180,E1 6600.565,E2 6600.565} C_VEL
LIN {X 0,Y 482.801,Z 733.66,A -85,B 0,C 180,E1 6602.327,E2 6602.327} C_VEL
LIN {X 0,Y 482.602,Z 733.66,A -85,B 0,C 180,E1 6608.864,E2 6608.864} C_VEL
LIN {X 0,Y 482.585,Z 733.66,A -85,B 0,C 180,E1 6613.809,E2 6613.809} C_VEL
LIN {X 0,Y 482.645,Z 733.66,A -85,B 0,C 180,E1 6618.842,E2 6618.842} C_VEL
LIN {X 0,Y 482.613,Z 733.66,A -85,B 0,C 180,E1 6624.656,E2 6624.656} C_VEL
LIN {X 0,Y 482.72,Z 733.66,A -85,B 0,C 180,E1 6629.874,E2 6629.874} C_VEL
LIN {X 0,Y 482.914,Z 733.66,A -85,B 0,C 180,E1 6635.943,E2 6635.943} C_VEL
LIN {X 0,Y 483.079,Z 733.66,A -85,B 0,C 180,E1 6641.731,E2 6641.731} C_VEL
LIN {X 0,Y 482.975,Z 733.66,A -85,B 0,C 180,E1 6647.32,E2 6647.32} C_VEL
LIN {X 0,Y 483.328,Z 733.66,A -85,B 0,C 180,E1 6652.798,E2 6652.798} C_VEL
LIN {X 0,Y 483.598,Z 733.66,A -85,B 0,C 180,E1 6658.202,E2 6658.202} C_VEL
LIN {X 0,Y 483.507,Z 733.66,A -85,B 0,C 180,E1 6663.587,E2 6663.587} C_VEL
LIN {X 0,Y 483.284,Z 733.66,A -85,B 0,C 180,E1 6669.008,E2 6669.008} C_VEL
LIN {X 0,Y 483.124,Z 733.66,A -85,B 0,C 180,E1 6674.515,E2 6674.515} C_VEL
LIN {X 0,Y 483.009,Z 733.66,A -85,B 0,C 180,E1 6680.165,E2 6680.165} C_VEL
LIN {X 0,Y 482.856,Z 733.66,A -85,B 0,C 180,E1 6686.034,E2 6686.034} C_VEL
LIN {X 0,Y 482.727,Z 733.66,A -85,B 0,C 180,E1 6692.216,E2 6692.216} C_VEL
LIN {X 0,Y 482.593,Z 733.66,A -85,B 0,C 180,E1 6698.857,E2 6698.857} C_VEL
LIN {X 0,Y 482.657,Z 733.66,A -85,B 0,C 180,E1 6703.82,E2 6703.82} C_VEL
LIN {X 0,Y 482.691,Z 733.66,A -85,B 0,C 180,E1 6708.826,E2 6708.826} C_VEL
LIN {X 0,Y 482.63,Z 733.66,A -85,B 0,C 180,E1 6712.165,E2 6712.165} C_VEL
LIN {X 0,Y 478.58,Z 732.146,A -85,B 0,C 180,E1 6713.555,E2 6713.555} C_VEL
LIN {X 0,Y 474.996,Z 732.942,A -85,B 0,C 180,E1 6714.615,E2 6714.615} C_VEL
LIN {X 0,Y 474.861,Z 733.944,A -85,B 0,C 180,E1 6714.845,E2 6714.845} C_VEL
LIN {X 0,Y 484.408,Z 767.947,A -85,B 0,C 180,E1 6717.902,E2 6717.902} C_VEL
LIN {X 0,Y 491.006,Z 780.877,A -85,B 0,C 180,E1 6718.598,E2 6718.598} C_VEL
LIN {X 0,Y 489.842,Z 822.107,A -85,B 0,C 180,E1 6719.435,E2 6719.435} C_VEL
LIN {X 0,Y 487.753,Z 857.35,A -85,B 0,C 180,E1 6720.794,E2 6720.794} C_VEL
LIN {X 0,Y 485.012,Z 893.598,A -85,B 0,C 180,E1 6722.973,E2 6722.973} C_VEL
LIN {X 0,Y 482.204,Z 926.106,A -85,B 0,C 180,E1 6725.777,E2 6725.777} C_VEL
LIN {X 0,Y 479.662,Z 957.196,A -85,B 0,C 180,E1 6729.336,E2 6729.336} C_VEL
LIN {X 0,Y 477.743,Z 981.961,A -85,B 0,C 180,E1 6733.211,E2 6733.211} C_VEL
LIN {X 0,Y 476.773,Z 998.523,A -85,B 0,C 180,E1 6736.707,E2 6736.707} C_VEL
LIN {X 0,Y 476.097,Z 1012.763,A -85,B 0,C 180,E1 6741.311,E2 6741.311} C_VEL
LIN {X 0,Y 475.85,Z 1020.141,A -85,B 0,C 180,E1 6745.437,E2 6745.437} C_VEL
LIN {X 0,Y 475.77,Z 1023,A -85,B 0,C 180,E1 6750,E2 6750} C_VEL
LIN {X 0,Y 475.893,Z 1020.147,A -85,B 0,C 180,E1 6754.562,E2 6754.562} C_VEL
LIN {X 0,Y 476.094,Z 1011.579,A -85,B 0,C 180,E1 6759.149,E2 6759.149} C_VEL
LIN {X 0,Y 476.74,Z 998.507,A -85,B 0,C 180,E1 6763.299,E2 6763.299} C_VEL
LIN {X 0,Y 477.766,Z 980.441,A -85,B 0,C 180,E1 6767.011,E2 6767.011} C_VEL
LIN {X 0,Y 479.537,Z 956.201,A -85,B 0,C 180,E1 6770.67,E2 6770.67} C_VEL
LIN {X 0,Y 482.084,Z 927.344,A -85,B 0,C 180,E1 6774.097,E2 6774.097} C_VEL
LIN {X 0,Y 484.924,Z 895.95,A -85,B 0,C 180,E1 6776.842,E2 6776.842} C_VEL
LIN {X 0,Y 487.644,Z 861.03,A -85,B 0,C 180,E1 6779.022,E2 6779.022} C_VEL
LIN {X 0,Y 489.771,Z 824.282,A -85,B 0,C 180,E1 6780.499,E2 6780.499} C_VEL
LIN {X 0,Y 490.998,Z 783.905,A -85,B 0,C 180,E1 6781.352,E2 6781.352} C_VEL
LIN {X 0,Y 490.396,Z 777.535,A -85,B 0,C 180,E1 6781.502,E2 6781.502} C_VEL
LIN {X 0,Y 480.969,Z 757.4,A -85,B 0,C 180,E1 6782.536,E2 6782.536} C_VEL
LIN {X 0,Y 477.023,Z 743.609,A -85,B 0,C 180,E1 6783.209,E2 6783.209} C_VEL
LIN {X 0,Y 474.846,Z 733.66,A -85,B 0,C 180,E1 6784.082,E2 6784.082} C_VEL
LIN {X 0,Y 474.684,Z 733.66,A -85,B 0,C 180,E1 6790.056,E2 6790.056} C_VEL
LIN {X 0,Y 474.678,Z 733.66,A -85,B 0,C 180,E1 6795.442,E2 6795.442} C_VEL
LIN {X 0,Y 474.62,Z 733.66,A -85,B 0,C 180,E1 6800.363,E2 6800.363} C_VEL
LIN {X 0,Y 474.749,Z 733.66,A -85,B 0,C 180,E1 6806.017,E2 6806.017} C_VEL
LIN {X 0,Y 474.806,Z 733.66,A -85,B 0,C 180,E1 6811.43,E2 6811.43} C_VEL
LIN {X 0,Y 474.987,Z 734.296,A -85,B 0,C 180,E1 6817.454,E2 6817.454} C_VEL
LIN {X 0,Y 482.355,Z 760.752,A -85,B 0,C 180,E1 6818.459,E2 6818.459} C_VEL
LIN {X 0,Y 481.954,Z 790.042,A -85,B 0,C 180,E1 6819.518,E2 6819.518} C_VEL
LIN {X 0,Y 480.968,Z 815.366,A -85,B 0,C 180,E1 6821.146,E2 6821.146} C_VEL
LIN {X 0,Y 479.712,Z 838.963,A -85,B 0,C 180,E1 6823.502,E2 6823.502} C_VEL
LIN {X 0,Y 478.526,Z 857.566,A -85,B 0,C 180,E1 6826.277,E2 6826.277} C_VEL
LIN {X 0,Y 477.613,Z 871.035,A -85,B 0,C 180,E1 6829.337,E2 6829.337} C_VEL
LIN {X 0,Y 477.076,Z 879.758,A -85,B 0,C 180,E1 6832.711,E2 6832.711} C_VEL
LIN {X 0,Y 476.734,Z 883.202,A -85,B 0,C 180,E1 6836.362,E2 6836.362} C_VEL
LIN {X 0,Y 476.754,Z 880.742,A -85,B 0,C 180,E1 6840.004,E2 6840.004} C_VEL
LIN {X 0,Y 477.088,Z 873.646,A -85,B 0,C 180,E1 6843.188,E2 6843.188} C_VEL
LIN {X 0,Y 477.633,Z 861.237,A -85,B 0,C 180,E1 6846.374,E2 6846.374} C_VEL
LIN {X 0,Y 478.581,Z 843.424,A -85,B 0,C 180,E1 6849.335,E2 6849.335} C_VEL
LIN {X 0,Y 479.693,Z 820.96,A -85,B 0,C 180,E1 6851.854,E2 6851.854} C_VEL
LIN {X 0,Y 480.977,Z 794.24,A -85,B 0,C 180,E1 6853.834,E2 6853.834} C_VEL
LIN {X 0,Y 481.766,Z 765.227,A -85,B 0,C 180,E1 6855.121,E2 6855.121} C_VEL
LIN {X 0,Y 481.028,Z 754.969,A -85,B 0,C 180,E1 6855.439,E2 6855.439} C_VEL
LIN {X 0,Y 475.173,Z 733.66,A -85,B 0,C 180,E1 6856.151,E2 6856.151} C_VEL
LIN {X 0,Y 474.997,Z 733.66,A -85,B 0,C 180,E1 6862.492,E2 6862.492} C_VEL
LIN {X 0,Y 474.788,Z 733.66,A -85,B 0,C 180,E1 6868.58,E2 6868.58} C_VEL
LIN {X 0,Y 474.713,Z 733.66,A -85,B 0,C 180,E1 6875.04,E2 6875.04} C_VEL
LIN {X 0,Y 474.619,Z 733.66,A -85,B 0,C 180,E1 6882.064,E2 6882.064} C_VEL
LIN {X 0,Y 474.702,Z 733.66,A -85,B 0,C 180,E1 6887.948,E2 6887.948} C_VEL
LIN {X 0,Y 474.721,Z 733.66,A -85,B 0,C 180,E1 6892.881,E2 6892.881} C_VEL
LIN {X 0,Y 474.842,Z 733.66,A -85,B 0,C 180,E1 6896.979,E2 6896.979} C_VEL
LIN {X 0,Y 491.278,Z 774.002,A -85,B 0,C 180,E1 6899.102,E2 6899.102} C_VEL
LIN {X 0,Y 489.17,Z 810.943,A -85,B 0,C 180,E1 6900.506,E2 6900.506} C_VEL
LIN {X 0,Y 486.383,Z 845.938,A -85,B 0,C 180,E1 6902.6,E2 6902.6} C_VEL
LIN {X 0,Y 483.245,Z 878.601,A -85,B 0,C 180,E1 6905.406,E2 6905.406} C_VEL
LIN {X 0,Y 480.427,Z 906.218,A -85,B 0,C 180,E1 6908.676,E2 6908.676} C_VEL
LIN {X 0,Y 478.162,Z 930.246,A -85,B 0,C 180,E1 6912.533,E2 6912.533} C_VEL
LIN {X 0,Y 476.773,Z 948.86,A -85,B 0,C 180,E1 6916.708,E2 6916.708} C_VEL
LIN {X 0,Y 476.051,Z 962.854,A -85,B 0,C 180,E1 6921.311,E2 6921.311} C_VEL
LIN {X 0,Y 475.801,Z 970.228,A -85,B 0,C 180,E1 6925.437,E2 6925.437} C_VEL
LIN {X 0,Y 475.816,Z 972.998,A -85,B 0,C 180,E1 6930,E2 6930} C_VEL
LIN {X 0,Y 475.881,Z 970.107,A -85,B 0,C 180,E1 6934.562,E2 6934.562} C_VEL
LIN {X 0,Y 476.075,Z 961.498,A -85,B 0,C 180,E1 6939.15,E2 6939.15} C_VEL
LIN {X 0,Y 476.829,Z 946.858,A -85,B 0,C 180,E1 6943.737,E2 6943.737} C_VEL
LIN {X 0,Y 478.267,Z 928.48,A -85,B 0,C 180,E1 6947.7,E2 6947.7} C_VEL
LIN {X 0,Y 480.472,Z 905.447,A -85,B 0,C 180,E1 6951.342,E2 6951.342} C_VEL
LIN {X 0,Y 483.459,Z 876.32,A -85,B 0,C 180,E1 6954.737,E2 6954.737} C_VEL
LIN {X 0,Y 486.506,Z 844.251,A -85,B 0,C 180,E1 6957.43,E2 6957.43} C_VEL
LIN {X 0,Y 489.311,Z 810.434,A -85,B 0,C 180,E1 6959.422,E2 6959.422} C_VEL
LIN {X 0,Y 491.38,Z 774.203,A -85,B 0,C 180,E1 6960.795,E2 6960.795} C_VEL
LIN {X 0,Y 478.257,Z 742.313,A -85,B 0,C 180,E1 6962.489,E2 6962.489} C_VEL
LIN {X 0,Y 474.879,Z 733.66,A -85,B 0,C 180,E1 6962.965,E2 6962.965} C_VEL
LIN {X 0,Y 474.61,Z 733.66,A -85,B 0,C 180,E1 6969.646,E2 6969.646} C_VEL
LIN {X 0,Y 474.632,Z 733.66,A -85,B 0,C 180,E1 6975.425,E2 6975.425} C_VEL
LIN {X 0,Y 474.657,Z 733.66,A -85,B 0,C 180,E1 6980.356,E2 6980.356} C_VEL
LIN {X 0,Y 474.681,Z 733.66,A -85,B 0,C 180,E1 6986.03,E2 6986.03} C_VEL
LIN {X 0,Y 474.815,Z 733.66,A -85,B 0,C 180,E1 6991.421,E2 6991.421} C_VEL
LIN {X 0,Y 475.051,Z 733.66,A -85,B 0,C 180,E1 6997.563,E2 6997.563} C_VEL
LIN {X 0,Y 475.098,Z 733.66,A -85,B 0,C 180,E1 7003.329,E2 7003.329} C_VEL
LIN {X 0,Y 475.171,Z 733.66,A -85,B 0,C 180,E1 7008.975,E2 7008.975} C_VEL
LIN {X 0,Y 475.463,Z 733.66,A -85,B 0,C 180,E1 7014.514,E2 7014.514} C_VEL
LIN {X 0,Y 475.619,Z 733.66,A -85,B 0,C 180,E1 7019.996,E2 7019.996} C_VEL
LIN {X 0,Y 475.425,Z 733.66,A -85,B 0,C 180,E1 7025.478,E2 7025.478} C_VEL
LIN {X 0,Y 475.289,Z 733.66,A -85,B 0,C 180,E1 7031.014,E2 7031.014} C_VEL
LIN {X 0,Y 475.11,Z 733.66,A -85,B 0,C 180,E1 7037.049,E2 7037.049} C_VEL
LIN {X 0,Y 475.016,Z 733.66,A -85,B 0,C 180,E1 7042.483,E2 7042.483} C_VEL
LIN {X 0,Y 474.826,Z 733.66,A -85,B 0,C 180,E1 7048.569,E2 7048.569} C_VEL
LIN {X 0,Y 474.709,Z 733.66,A -85,B 0,C 180,E1 7055.03,E2 7055.03} C_VEL
LIN {X 0,Y 474.631,Z 733.66,A -85,B 0,C 180,E1 7062.052,E2 7062.052} C_VEL
LIN {X 0,Y 474.692,Z 733.66,A -85,B 0,C 180,E1 7067.946,E2 7067.946} C_VEL
LIN {X 0,Y 474.861,Z 733.944,A -85,B 0,C 180,E1 7074.845,E2 7074.845} C_VEL
LIN {X 0,Y 474.122,Z 757.939,A -85,B 0,C 180,E1 7076.643,E2 7076.643} C_VEL
LIN {X 0,Y 474.955,Z 763.644,A -85,B 0,C 180,E1 7077.11,E2 7077.11} C_VEL
LIN {X 0,Y 484.187,Z 782.388,A -85,B 0,C 180,E1 7078.132,E2 7078.132} C_VEL
LIN {X 0,Y 482.92,Z 824.226,A -85,B 0,C 180,E1 7079.029,E2 7079.029} C_VEL
LIN {X 0,Y 480.524,Z 861.123,A -85,B 0,C 180,E1 7080.532,E2 7080.532} C_VEL
LIN {X 0,Y 477.528,Z 896.527,A -85,B 0,C 180,E1 7082.787,E2 7082.787} C_VEL
LIN {X 0,Y 474.589,Z 928.107,A -85,B 0,C 180,E1 7085.622,E2 7085.622} C_VEL
LIN {X 0,Y 471.871,Z 956.523,A -85,B 0,C 180,E1 7089.086,E2 7089.086} C_VEL
LIN {X 0,Y 469.87,Z 981.866,A -85,B 0,C 180,E1 7093.141,E2 7093.141} C_VEL
LIN {X 0,Y 468.801,Z 999.126,A -85,B 0,C 180,E1 7096.933,E2 7096.933} C_VEL
LIN {X 0,Y 468.223,Z 1012.566,A -85,B 0,C 180,E1 7101.164,E2 7101.164} C_VEL
LIN {X 0,Y 467.953,Z 1020.137,A -85,B 0,C 180,E1 7105.36,E2 7105.36} C_VEL
LIN {X 0,Y 467.878,Z 1023,A -85,B 0,C 180,E1 7110,E2 7110} C_VEL
LIN {X 0,Y 468.015,Z 1020.142,A -85,B 0,C 180,E1 7114.639,E2 7114.639} C_VEL
LIN {X 0,Y 468.227,Z 1012.557,A -85,B 0,C 180,E1 7118.835,E2 7118.835} C_VEL
LIN {X 0,Y 468.783,Z 998.934,A -85,B 0,C 180,E1 7123.067,E2 7123.067} C_VEL
LIN {X 0,Y 469.832,Z 981.186,A -85,B 0,C 180,E1 7126.86,E2 7126.86} C_VEL
LIN {X 0,Y 472.012,Z 954.712,A -85,B 0,C 180,E1 7131.169,E2 7131.169} C_VEL
LIN {X 0,Y 474.801,Z 925.915,A -85,B 0,C 180,E1 7134.602,E2 7134.602} C_VEL
LIN {X 0,Y 477.93,Z 893.591,A -85,B 0,C 180,E1 7137.431,E2 7137.431} C_VEL
LIN {X 0,Y 480.787,Z 859.397,A -85,B 0,C 180,E1 7139.545,E2 7139.545} C_VEL
LIN {X 0,Y 482.969,Z 823.529,A -85,B 0,C 180,E1 7140.991,E2 7140.991} C_VEL
LIN {X 0,Y 484.045,Z 781.263,A -85,B 0,C 180,E1 7141.897,E2 7141.897} C_VEL
LIN {X 0,Y 474.077,Z 758.594,A -85,B 0,C 180,E1 7143.044,E2 7143.044} C_VEL
LIN {X 0,Y 468.396,Z 740.142,A -85,B 0,C 180,E1 7143.91,E2 7143.91} C_VEL
LIN {X 0,Y 466.907,Z 733.66,A -85,B 0,C 180,E1 7144.49,E2 7144.49} C_VEL
LIN {X 0,Y 466.749,Z 733.66,A -85,B 0,C 180,E1 7150.45,E2 7150.45} C_VEL
LIN {X 0,Y 466.762,Z 733.66,A -85,B 0,C 180,E1 7157.071,E2 7157.071} C_VEL
LIN {X 0,Y 466.752,Z 733.66,A -85,B 0,C 180,E1 7164.191,E2 7164.191} C_VEL
LIN {X 0,Y 466.844,Z 733.66,A -85,B 0,C 180,E1 7168.747,E2 7168.747} C_VEL
LIN {X 0,Y 466.956,Z 733.66,A -85,B 0,C 180,E1 7175.215,E2 7175.215} C_VEL
LIN {X 0,Y 467.045,Z 734.02,A -85,B 0,C 180,E1 7176.965,E2 7176.965} C_VEL
LIN {X 0,Y 475.077,Z 762.19,A -85,B 0,C 180,E1 7178.126,E2 7178.126} C_VEL
LIN {X 0,Y 474.647,Z 791.471,A -85,B 0,C 180,E1 7179.205,E2 7179.205} C_VEL
LIN {X 0,Y 473.584,Z 816.538,A -85,B 0,C 180,E1 7180.841,E2 7180.841} C_VEL
LIN {X 0,Y 472.242,Z 840.165,A -85,B 0,C 180,E1 7183.234,E2 7183.234} C_VEL
LIN {X 0,Y 470.957,Z 858.804,A -85,B 0,C 180,E1 7186.052,E2 7186.052} C_VEL
LIN {X 0,Y 469.945,Z 872.394,A -85,B 0,C 180,E1 7189.195,E2 7189.195} C_VEL
LIN {X 0,Y 469.318,Z 881.021,A -85,B 0,C 180,E1 7192.59,E2 7192.59} C_VEL
LIN {X 0,Y 468.972,Z 884.477,A -85,B 0,C 180,E1 7196.302,E2 7196.302} C_VEL
LIN {X 0,Y 468.963,Z 882.012,A -85,B 0,C 180,E1 7200.004,E2 7200.004} C_VEL
LIN {X 0,Y 469.309,Z 874.915,A -85,B 0,C 180,E1 7203.241,E2 7203.241} C_VEL
LIN {X 0,Y 469.907,Z 862.502,A -85,B 0,C 180,E1 7206.479,E2 7206.479} C_VEL
LIN {X 0,Y 470.911,Z 844.712,A -85,B 0,C 180,E1 7209.488,E2 7209.488} C_VEL
LIN {X 0,Y 472.088,Z 822.332,A -85,B 0,C 180,E1 7212.044,E2 7212.044} C_VEL
LIN {X 0,Y 473.389,Z 796.688,A -85,B 0,C 180,E1 7214.001,E2 7214.001} C_VEL
LIN {X 0,Y 474.213,Z 768.718,A -85,B 0,C 180,E1 7215.317,E2 7215.317} C_VEL
LIN {X 0,Y 473.555,Z 756.501,A -85,B 0,C 180,E1 7215.709,E2 7215.709} C_VEL
LIN {X 0,Y 467.241,Z 733.66,A -85,B 0,C 180,E1 7216.483,E2 7216.483} C_VEL
LIN {X 0,Y 467.043,Z 733.66,A -85,B 0,C 180,E1 7222.897,E2 7222.897} C_VEL
LIN {X 0,Y 466.851,Z 733.66,A -85,B 0,C 180,E1 7229.112,E2 7229.112} C_VEL
LIN {X 0,Y 466.736,Z 733.66,A -85,B 0,C 180,E1 7235.73,E2 7235.73} C_VEL
LIN {X 0,Y 466.677,Z 733.66,A -85,B 0,C 180,E1 7241.737,E2 7241.737} C_VEL
LIN {X 0,Y 466.79,Z 733.66,A -85,B 0,C 180,E1 7248.251,E2 7248.251} C_VEL
LIN {X 0,Y 466.746,Z 733.66,A -85,B 0,C 180,E1 7254.274,E2 7254.274} C_VEL
LIN {X 0,Y 466.885,Z 733.66,A -85,B 0,C 180,E1 7256.341,E2 7256.341} C_VEL
LIN {X 0,Y 484.399,Z 775.488,A -85,B 0,C 180,E1 7258.654,E2 7258.654} C_VEL
LIN {X 0,Y 482.211,Z 812.442,A -85,B 0,C 180,E1 7260.102,E2 7260.102} C_VEL
LIN {X 0,Y 479.321,Z 846.653,A -85,B 0,C 180,E1 7262.189,E2 7262.189} C_VEL
LIN {X 0,Y 475.971,Z 878.984,A -85,B 0,C 180,E1 7265.004,E2 7265.004} C_VEL
LIN {X 0,Y 472.941,Z 906.809,A -85,B 0,C 180,E1 7268.349,E2 7268.349} C_VEL
LIN {X 0,Y 470.566,Z 930.105,A -85,B 0,C 180,E1 7272.139,E2 7272.139} C_VEL
LIN {X 0,Y 469.096,Z 948.229,A -85,B 0,C 180,E1 7276.193,E2 7276.193} C_VEL
LIN {X 0,Y 468.242,Z 961.951,A -85,B 0,C 180,E1 7280.696,E2 7280.696} C_VEL
LIN {X 0,Y 467.917,Z 970.245,A -85,B 0,C 180,E1 7285.36,E2 7285.36} C_VEL
LIN {X 0,Y 467.926,Z 972.998,A -85,B 0,C 180,E1 7290,E2 7290} C_VEL
LIN {X 0,Y 467.984,Z 970.126,A -85,B 0,C 180,E1 7294.64,E2 7294.64} C_VEL
LIN {X 0,Y 468.22,Z 961.743,A -85,B 0,C 180,E1 7299.305,E2 7299.305} C_VEL
LIN {X 0,Y 469.042,Z 947.906,A -85,B 0,C 180,E1 7303.808,E2 7303.808} C_VEL
LIN {X 0,Y 470.616,Z 929.196,A -85,B 0,C 180,E1 7307.94,E2 7307.94} C_VEL
LIN {X 0,Y 472.983,Z 906.06,A -85,B 0,C 180,E1 7311.667,E2 7311.667} C_VEL
LIN {X 0,Y 476.095,Z 877.865,A -85,B 0,C 180,E1 7315.024,E2 7315.024} C_VEL
LIN {X 0,Y 479.332,Z 846.218,A -85,B 0,C 180,E1 7317.753,E2 7317.753} C_VEL
LIN {X 0,Y 482.363,Z 811.961,A -85,B 0,C 180,E1 7319.823,E2 7319.823} C_VEL
LIN {X 0,Y 484.183,Z 774.28,A -85,B 0,C 180,E1 7321.311,E2 7321.311} C_VEL
LIN {X 0,Y 466.917,Z 733.66,A -85,B 0,C 180,E1 7323.593,E2 7323.593} C_VEL
LIN {X 0,Y 466.661,Z 733.66,A -85,B 0,C 180,E1 7330.459,E2 7330.459} C_VEL
LIN {X 0,Y 466.758,Z 733.66,A -85,B 0,C 180,E1 7337.059,E2 7337.059} C_VEL
LIN {X 0,Y 466.717,Z 733.66,A -85,B 0,C 180,E1 7341.945,E2 7341.945} C_VEL
LIN {X 0,Y 466.778,Z 733.66,A -85,B 0,C 180,E1 7348.732,E2 7348.732} C_VEL
LIN {X 0,Y 467.077,Z 733.66,A -85,B 0,C 180,E1 7355.184,E2 7355.184} C_VEL
LIN {X 0,Y 467.214,Z 733.66,A -85,B 0,C 180,E1 7361.088,E2 7361.088} C_VEL
LIN {X 0,Y 467.132,Z 733.66,A -85,B 0,C 180,E1 7366.883,E2 7366.883} C_VEL
LIN {X 0,Y 467.477,Z 733.66,A -85,B 0,C 180,E1 7372.552,E2 7372.552} C_VEL
LIN {X 0,Y 467.784,Z 733.66,A -85,B 0,C 180,E1 7378.141,E2 7378.141} C_VEL
LIN {X 0,Y 467.707,Z 733.66,A -85,B 0,C 180,E1 7383.708,E2 7383.708} C_VEL
LIN {X 0,Y 467.462,Z 733.66,A -85,B 0,C 180,E1 7389.315,E2 7389.315} C_VEL
LIN {X 0,Y 467.253,Z 733.66,A -85,B 0,C 180,E1 7395.019,E2 7395.019} C_VEL
LIN {X 0,Y 467.123,Z 733.66,A -85,B 0,C 180,E1 7400.882,E2 7400.882} C_VEL
LIN {X 0,Y 466.941,Z 733.66,A -85,B 0,C 180,E1 7406.992,E2 7406.992} C_VEL
LIN {X 0,Y 466.801,Z 733.66,A -85,B 0,C 180,E1 7413.456,E2 7413.456} C_VEL
LIN {X 0,Y 466.677,Z 733.66,A -85,B 0,C 180,E1 7420.449,E2 7420.449} C_VEL
LIN {X 0,Y 466.805,Z 733.66,A -85,B 0,C 180,E1 7427.067,E2 7427.067} C_VEL
LIN {X 0,Y 466.871,Z 733.66,A -85,B 0,C 180,E1 7434.159,E2 7434.159} C_VEL
LIN {X 0,Y 473.582,Z 758.366,A -85,B 0,C 180,E1 7436.642,E2 7436.642} C_VEL
LIN {X 0,Y 474.955,Z 763.644,A -85,B 0,C 180,E1 7437.11,E2 7437.11} C_VEL
LIN {X 0,Y 477.86,Z 776.007,A -85,B 0,C 180,E1 7437.552,E2 7437.552} C_VEL
LIN {X 0,Y 477.276,Z 798.399,A -85,B 0,C 180,E1 7437.914,E2 7437.914} C_VEL
LIN {X 0,Y 475.374,Z 835.35,A -85,B 0,C 180,E1 7438.923,E2 7438.923} C_VEL
LIN {X 0,Y 472.662,Z 871.824,A -85,B 0,C 180,E1 7440.676,E2 7440.676} C_VEL
LIN {X 0,Y 469.354,Z 906.171,A -85,B 0,C 180,E1 7443.152,E2 7443.152} C_VEL
LIN {X 0,Y 466.162,Z 937.561,A -85,B 0,C 180,E1 7446.31,E2 7446.31} C_VEL
LIN {X 0,Y 463.555,Z 964.096,A -85,B 0,C 180,E1 7449.943,E2 7449.943} C_VEL
LIN {X 0,Y 461.524,Z 988.914,A -85,B 0,C 180,E1 7454.541,E2 7454.541} C_VEL
LIN {X 0,Y 460.561,Z 1004.648,A -85,B 0,C 180,E1 7458.624,E2 7458.624} C_VEL
LIN {X 0,Y 460.226,Z 1014.668,A -85,B 0,C 180,E1 7462.438,E2 7462.438} C_VEL
LIN {X 0,Y 460.045,Z 1020.516,A -85,B 0,C 180,E1 7466.226,E2 7466.226} C_VEL
LIN {X 0,Y 459.996,Z 1022.458,A -85,B 0,C 180,E1 7470,E2 7470} C_VEL
LIN {X 0,Y 460.068,Z 1020.484,A -85,B 0,C 180,E1 7473.774,E2 7473.774} C_VEL
LIN {X 0,Y 460.345,Z 1012.522,A -85,B 0,C 180,E1 7478.495,E2 7478.495} C_VEL
LIN {X 0,Y 460.853,Z 999.27,A -85,B 0,C 180,E1 7482.812,E2 7482.812} C_VEL
LIN {X 0,Y 462.186,Z 978.892,A -85,B 0,C 180,E1 7487.459,E2 7487.459} C_VEL
LIN {X 0,Y 464.408,Z 954.909,A -85,B 0,C 180,E1 7491.447,E2 7491.447} C_VEL
LIN {X 0,Y 467.33,Z 926.554,A -85,B 0,C 180,E1 7494.909,E2 7494.909} C_VEL
LIN {X 0,Y 470.634,Z 894.61,A -85,B 0,C 180,E1 7497.775,E2 7497.775} C_VEL
LIN {X 0,Y 473.805,Z 859.614,A -85,B 0,C 180,E1 7499.994,E2 7499.994} C_VEL
LIN {X 0,Y 476.188,Z 823.228,A -85,B 0,C 180,E1 7501.482,E2 7501.482} C_VEL
LIN {X 0,Y 476.901,Z 783.397,A -85,B 0,C 180,E1 7502.392,E2 7502.392} C_VEL
LIN {X 0,Y 466.743,Z 758.446,A -85,B 0,C 180,E1 7503.63,E2 7503.63} C_VEL
LIN {X 0,Y 459.507,Z 736.449,A -85,B 0,C 180,E1 7504.714,E2 7504.714} C_VEL
LIN {X 0,Y 458.945,Z 733.66,A -85,B 0,C 180,E1 7505.031,E2 7505.031} C_VEL
LIN {X 0,Y 458.865,Z 733.66,A -85,B 0,C 180,E1 7511.294,E2 7511.294} C_VEL
LIN {X 0,Y 458.834,Z 733.66,A -85,B 0,C 180,E1 7516.549,E2 7516.549} C_VEL
LIN {X 0,Y 458.766,Z 733.66,A -85,B 0,C 180,E1 7522.381,E2 7522.381} C_VEL
LIN {X 0,Y 458.934,Z 733.66,A -85,B 0,C 180,E1 7529.068,E2 7529.068} C_VEL
LIN {X 0,Y 459.093,Z 733.66,A -85,B 0,C 180,E1 7535.827,E2 7535.827} C_VEL
LIN {X 0,Y 459.171,Z 734.488,A -85,B 0,C 180,E1 7536.455,E2 7536.455} C_VEL
LIN {X 0,Y 467.821,Z 761.909,A -85,B 0,C 180,E1 7537.728,E2 7537.728} C_VEL
LIN {X 0,Y 467.476,Z 789.7,A -85,B 0,C 180,E1 7538.713,E2 7538.713} C_VEL
LIN {X 0,Y 466.264,Z 817.509,A -85,B 0,C 180,E1 7540.502,E2 7540.502} C_VEL
LIN {X 0,Y 464.963,Z 839.535,A -85,B 0,C 180,E1 7542.719,E2 7542.719} C_VEL
LIN {X 0,Y 463.477,Z 858.761,A -85,B 0,C 180,E1 7545.581,E2 7545.581} C_VEL
LIN {X 0,Y 462.377,Z 872.525,A -85,B 0,C 180,E1 7548.674,E2 7548.674} C_VEL
LIN {X 0,Y 461.661,Z 880.495,A -85,B 0,C 180,E1 7551.518,E2 7551.518} C_VEL
LIN {X 0,Y 461.423,Z 884.764,A -85,B 0,C 180,E1 7554.355,E2 7554.355} C_VEL
LIN {X 0,Y 461.152,Z 885.241,A -85,B 0,C 180,E1 7558.123,E2 7558.123} C_VEL
LIN {X 0,Y 461.328,Z 879.826,A -85,B 0,C 180,E1 7561.885,E2 7561.885} C_VEL
LIN {X 0,Y 461.851,Z 869.811,A -85,B 0,C 180,E1 7565.176,E2 7565.176} C_VEL
LIN {X 0,Y 462.731,Z 853.634,A -85,B 0,C 180,E1 7568.471,E2 7568.471} C_VEL
LIN {X 0,Y 463.992,Z 832.809,A -85,B 0,C 180,E1 7571.295,E2 7571.295} C_VEL
LIN {X 0,Y 465.342,Z 808.392,A -85,B 0,C 180,E1 7573.528,E2 7573.528} C_VEL
LIN {X 0,Y 466.428,Z 781.137,A -85,B 0,C 180,E1 7575.136,E2 7575.136} C_VEL
LIN {X 0,Y 466.191,Z 758.484,A -85,B 0,C 180,E1 7575.964,E2 7575.964} C_VEL
LIN {X 0,Y 459.308,Z 733.66,A -85,B 0,C 180,E1 7576.842,E2 7576.842} C_VEL
LIN {X 0,Y 459.104,Z 733.66,A -85,B 0,C 180,E1 7583.316,E2 7583.316} C_VEL
LIN {X 0,Y 458.875,Z 733.66,A -85,B 0,C 180,E1 7589.669,E2 7589.669} C_VEL
LIN {X 0,Y 458.761,Z 733.66,A -85,B 0,C 180,E1 7596.449,E2 7596.449} C_VEL
LIN {X 0,Y 458.837,Z 733.66,A -85,B 0,C 180,E1 7603.451,E2 7603.451} C_VEL
LIN {X 0,Y 458.876,Z 733.66,A -85,B 0,C 180,E1 7609.37,E2 7609.37} C_VEL
LIN {X 0,Y 458.938,Z 733.669,A -85,B 0,C 180,E1 7615.694,E2 7615.694} C_VEL
LIN {X 0,Y 477.284,Z 776.834,A -85,B 0,C 180,E1 7618.17,E2 7618.17} C_VEL
LIN {X 0,Y 475.268,Z 813.95,A -85,B 0,C 180,E1 7619.686,E2 7619.686} C_VEL
LIN {X 0,Y 472.148,Z 848.74,A -85,B 0,C 180,E1 7621.865,E2 7621.865} C_VEL
LIN {X 0,Y 468.704,Z 879.64,A -85,B 0,C 180,E1 7624.621,E2 7624.621} C_VEL
LIN {X 0,Y 465.5,Z 907.202,A -85,B 0,C 180,E1 7627.985,E2 7627.985} C_VEL
LIN {X 0,Y 462.922,Z 930.847,A -85,B 0,C 180,E1 7631.899,E2 7631.899} C_VEL
LIN {X 0,Y 461.308,Z 948.976,A -85,B 0,C 180,E1 7636.054,E2 7636.054} C_VEL
LIN {X 0,Y 460.384,Z 962.567,A -85,B 0,C 180,E1 7640.626,E2 7640.626} C_VEL
LIN {X 0,Y 460.041,Z 970.651,A -85,B 0,C 180,E1 7645.281,E2 7645.281} C_VEL
LIN {X 0,Y 460.033,Z 973.345,A -85,B 0,C 180,E1 7650,E2 7650} C_VEL
LIN {X 0,Y 460.099,Z 970.534,A -85,B 0,C 180,E1 7654.719,E2 7654.719} C_VEL
LIN {X 0,Y 460.4,Z 962.152,A -85,B 0,C 180,E1 7659.465,E2 7659.465} C_VEL
LIN {X 0,Y 461.252,Z 948.685,A -85,B 0,C 180,E1 7663.944,E2 7663.944} C_VEL
LIN {X 0,Y 463.134,Z 928.899,A -85,B 0,C 180,E1 7668.375,E2 7668.375} C_VEL
LIN {X 0,Y 465.75,Z 904.957,A -85,B 0,C 180,E1 7672.243,E2 7672.243} C_VEL
LIN {X 0,Y 469.172,Z 876.024,A -85,B 0,C 180,E1 7675.656,E2 7675.656} C_VEL
LIN {X 0,Y 472.552,Z 844.343,A -85,B 0,C 180,E1 7678.364,E2 7678.364} C_VEL
LIN {X 0,Y 475.688,Z 809.973,A -85,B 0,C 180,E1 7680.417,E2 7680.417} C_VEL
LIN {X 0,Y 477.081,Z 775.837,A -85,B 0,C 180,E1 7681.791,E2 7681.791} C_VEL
LIN {X 0,Y 460.347,Z 738.044,A -85,B 0,C 180,E1 7684.012,E2 7684.012} C_VEL
LIN {X 0,Y 458.947,Z 733.66,A -85,B 0,C 180,E1 7684.362,E2 7684.362} C_VEL
LIN {X 0,Y 458.728,Z 733.66,A -85,B 0,C 180,E1 7691.31,E2 7691.31} C_VEL
LIN {X 0,Y 458.829,Z 733.66,A -85,B 0,C 180,E1 7696.551,E2 7696.551} C_VEL
LIN {X 0,Y 458.786,Z 733.66,A -85,B 0,C 180,E1 7702.378,E2 7702.378} C_VEL
LIN {X 0,Y 458.864,Z 733.66,A -85,B 0,C 180,E1 7709.083,E2 7709.083} C_VEL
LIN {X 0,Y 459.082,Z 733.66,A -85,B 0,C 180,E1 7714.609,E2 7714.609} C_VEL
LIN {X 0,Y 459.309,Z 733.66,A -85,B 0,C 180,E1 7720.749,E2 7720.749} C_VEL
LIN {X 0,Y 459.231,Z 733.66,A -85,B 0,C 180,E1 7726.653,E2 7726.653} C_VEL
LIN {X 0,Y 459.551,Z 733.66,A -85,B 0,C 180,E1 7732.423,E2 7732.423} C_VEL
LIN {X 0,Y 459.872,Z 733.66,A -85,B 0,C 180,E1 7738.109,E2 7738.109} C_VEL
LIN {X 0,Y 459.79,Z 733.66,A -85,B 0,C 180,E1 7743.772,E2 7743.772} C_VEL
LIN {X 0,Y 459.549,Z 733.66,A -85,B 0,C 180,E1 7749.477,E2 7749.477} C_VEL
LIN {X 0,Y 459.32,Z 733.66,A -85,B 0,C 180,E1 7755.285,E2 7755.285} C_VEL
LIN {X 0,Y 459.168,Z 733.66,A -85,B 0,C 180,E1 7761.262,E2 7761.262} C_VEL
LIN {X 0,Y 458.992,Z 733.66,A -85,B 0,C 180,E1 7767.498,E2 7767.498} C_VEL
LIN {X 0,Y 458.807,Z 733.66,A -85,B 0,C 180,E1 7774.118,E2 7774.118} C_VEL
LIN {X 0,Y 458.785,Z 733.66,A -85,B 0,C 180,E1 7780.619,E2 7780.619} C_VEL
LIN {X 0,Y 458.863,Z 733.66,A -85,B 0,C 180,E1 7786.536,E2 7786.536} C_VEL
LIN {X 0,Y 458.836,Z 733.66,A -85,B 0,C 180,E1 7792.358,E2 7792.358} C_VEL
LIN {X 0,Y 458.9,Z 733.737,A -85,B 0,C 180,E1 7793.749,E2 7793.749} C_VEL
LIN {X 0,Y 467.048,Z 762.833,A -85,B 0,C 180,E1 7796.476,E2 7796.476} C_VEL
LIN {X 0,Y 477.488,Z 787.39,A -85,B 0,C 180,E1 7797.722,E2 7797.722} C_VEL
LIN {X 0,Y 477.276,Z 798.399,A -85,B 0,C 180,E1 7797.914,E2 7797.914} C_VEL
LIN {X 0,Y 473.109,Z 815.451,A -85,B 0,C 180,E1 7798.032,E2 7798.032} C_VEL
LIN {X 0,Y 468.943,Z 830.178,A -85,B 0,C 180,E1 7798.247,E2 7798.247} C_VEL
LIN {X 0,Y 468.755,Z 832.219,A -85,B 0,C 180,E1 7798.318,E2 7798.318} C_VEL
LIN {X 0,Y 466.005,Z 867.784,A -85,B 0,C 180,E1 7799.981,E2 7799.981} C_VEL
LIN {X 0,Y 462.533,Z 902.656,A -85,B 0,C 180,E1 7802.428,E2 7802.428} C_VEL
LIN {X 0,Y 459.082,Z 933.929,A -85,B 0,C 180,E1 7805.527,E2 7805.527} C_VEL
LIN {X 0,Y 456.252,Z 960.573,A -85,B 0,C 180,E1 7809.099,E2 7809.099} C_VEL
LIN {X 0,Y 454.013,Z 983.598,A -85,B 0,C 180,E1 7813.283,E2 7813.283} C_VEL
LIN {X 0,Y 452.817,Z 1001.99,A -85,B 0,C 180,E1 7817.937,E2 7817.937} C_VEL
LIN {X 0,Y 452.386,Z 1013.588,A -85,B 0,C 180,E1 7822.306,E2 7822.306} C_VEL
LIN {X 0,Y 452.209,Z 1019.458,A -85,B 0,C 180,E1 7826.16,E2 7826.16} C_VEL
LIN {X 0,Y 452.168,Z 1021.388,A -85,B 0,C 180,E1 7830,E2 7830} C_VEL
LIN {X 0,Y 452.256,Z 1019.359,A -85,B 0,C 180,E1 7833.839,E2 7833.839} C_VEL
LIN {X 0,Y 452.505,Z 1011.545,A -85,B 0,C 180,E1 7838.513,E2 7838.513} C_VEL
LIN {X 0,Y 453.137,Z 996.684,A -85,B 0,C 180,E1 7843.526,E2 7843.526} C_VEL
LIN {X 0,Y 454.449,Z 978.662,A -85,B 0,C 180,E1 7847.728,E2 7847.728} C_VEL
LIN {X 0,Y 456.8,Z 954.949,A -85,B 0,C 180,E1 7851.755,E2 7851.755} C_VEL
LIN {X 0,Y 460.033,Z 926.162,A -85,B 0,C 180,E1 7855.332,E2 7855.332} C_VEL
LIN {X 0,Y 463.409,Z 895.278,A -85,B 0,C 180,E1 7858.157,E2 7858.157} C_VEL
LIN {X 0,Y 466.79,Z 860.408,A -85,B 0,C 180,E1 7860.426,E2 7860.426} C_VEL
LIN {X 0,Y 469.381,Z 823.738,A -85,B 0,C 180,E1 7861.964,E2 7861.964} C_VEL
LIN {X 0,Y 470.242,Z 786.223,A -85,B 0,C 180,E1 7862.855,E2 7862.855} C_VEL
LIN {X 0,Y 460.185,Z 760.486,A -85,B 0,C 180,E1 7864.133,E2 7864.133} C_VEL
LIN {X 0,Y 451.014,Z 733.66,A -85,B 0,C 180,E1 7865.504,E2 7865.504} C_VEL
LIN {X 0,Y 450.881,Z 733.66,A -85,B 0,C 180,E1 7872.383,E2 7872.383} C_VEL
LIN {X 0,Y 450.832,Z 733.66,A -85,B 0,C 180,E1 7877.811,E2 7877.811} C_VEL
LIN {X 0,Y 450.877,Z 733.66,A -85,B 0,C 180,E1 7883.701,E2 7883.701} C_VEL
LIN {X 0,Y 450.984,Z 733.66,A -85,B 0,C 180,E1 7889.769,E2 7889.769} C_VEL
LIN {X 0,Y 451.203,Z 733.66,A -85,B 0,C 180,E1 7895.843,E2 7895.843} C_VEL
LIN {X 0,Y 460.536,Z 763.101,A -85,B 0,C 180,E1 7897.339,E2 7897.339} C_VEL
LIN {X 0,Y 460.235,Z 791.369,A -85,B 0,C 180,E1 7898.369,E2 7898.369} C_VEL
LIN {X 0,Y 459.002,Z 818.112,A -85,B 0,C 180,E1 7900.118,E2 7900.118} C_VEL
LIN {X 0,Y 457.543,Z 840.897,A -85,B 0,C 180,E1 7902.43,E2 7902.43} C_VEL
LIN {X 0,Y 455.93,Z 860.087,A -85,B 0,C 180,E1 7905.337,E2 7905.337} C_VEL
LIN {X 0,Y 454.717,Z 873.821,A -85,B 0,C 180,E1 7908.481,E2 7908.481} C_VEL
LIN {X 0,Y 453.929,Z 881.809,A -85,B 0,C 180,E1 7911.372,E2 7911.372} C_VEL
LIN {X 0,Y 453.671,Z 886.054,A -85,B 0,C 180,E1 7914.258,E2 7914.258} C_VEL
LIN {X 0,Y 453.367,Z 886.521,A -85,B 0,C 180,E1 7918.091,E2 7918.091} C_VEL
LIN {X 0,Y 453.541,Z 881.081,A -85,B 0,C 180,E1 7921.917,E2 7921.917} C_VEL
LIN {X 0,Y 454.083,Z 871.049,A -85,B 0,C 180,E1 7925.265,E2 7925.265} C_VEL
LIN {X 0,Y 455.015,Z 854.869,A -85,B 0,C 180,E1 7928.616,E2 7928.616} C_VEL
LIN {X 0,Y 456.34,Z 834.052,A -85,B 0,C 180,E1 7931.487,E2 7931.487} C_VEL
LIN {X 0,Y 457.766,Z 809.707,A -85,B 0,C 180,E1 7933.756,E2 7933.756} C_VEL
LIN {X 0,Y 458.937,Z 780.841,A -85,B 0,C 180,E1 7935.474,E2 7935.474} C_VEL
LIN {X 0,Y 458.572,Z 759.463,A -85,B 0,C 180,E1 7936.265,E2 7936.265} C_VEL
LIN {X 0,Y 451.379,Z 733.66,A -85,B 0,C 180,E1 7937.168,E2 7937.168} C_VEL
LIN {X 0,Y 451.135,Z 733.66,A -85,B 0,C 180,E1 7943.753,E2 7943.753} C_VEL
LIN {X 0,Y 450.949,Z 733.66,A -85,B 0,C 180,E1 7950.244,E2 7950.244} C_VEL
LIN {X 0,Y 450.835,Z 733.66,A -85,B 0,C 180,E1 7957.197,E2 7957.197} C_VEL
LIN {X 0,Y 450.815,Z 733.66,A -85,B 0,C 180,E1 7962.364,E2 7962.364} C_VEL
LIN {X 0,Y 450.901,Z 733.66,A -85,B 0,C 180,E1 7967.811,E2 7967.811} C_VEL
LIN {X 0,Y 450.917,Z 733.66,A -85,B 0,C 180,E1 7974.604,E2 7974.604} C_VEL
LIN {X 0,Y 450.955,Z 733.66,A -85,B 0,C 180,E1 7974.975,E2 7974.975} C_VEL
LIN {X 0,Y 469.988,Z 777.75,A -85,B 0,C 180,E1 7977.637,E2 7977.637} C_VEL
LIN {X 0,Y 470.354,Z 789.134,A -85,B 0,C 180,E1 7978.097,E2 7978.097} C_VEL
LIN {X 0,Y 467.711,Z 823.621,A -85,B 0,C 180,E1 7979.711,E2 7979.711} C_VEL
LIN {X 0,Y 464.317,Z 856.409,A -85,B 0,C 180,E1 7981.988,E2 7981.988} C_VEL
LIN {X 0,Y 460.533,Z 888.088,A -85,B 0,C 180,E1 7985.088,E2 7985.088} C_VEL
LIN {X 0,Y 457.256,Z 914.442,A -85,B 0,C 180,E1 7988.64,E2 7988.64} C_VEL
LIN {X 0,Y 454.649,Z 937.144,A -85,B 0,C 180,E1 7992.809,E2 7992.809} C_VEL
LIN {X 0,Y 453.17,Z 953.368,A -85,B 0,C 180,E1 7996.967,E2 7996.967} C_VEL
LIN {X 0,Y 452.423,Z 965.264,A -85,B 0,C 180,E1 8001.51,E2 8001.51} C_VEL
LIN {X 0,Y 452.139,Z 972.01,A -85,B 0,C 180,E1 8006.16,E2 8006.16} C_VEL
LIN {X 0,Y 452.143,Z 973.751,A -85,B 0,C 180,E1 8010,E2 8010} C_VEL
LIN {X 0,Y 452.235,Z 970.941,A -85,B 0,C 180,E1 8014.802,E2 8014.802} C_VEL
LIN {X 0,Y 452.574,Z 962.561,A -85,B 0,C 180,E1 8019.63,E2 8019.63} C_VEL
LIN {X 0,Y 453.465,Z 949.581,A -85,B 0,C 180,E1 8024.045,E2 8024.045} C_VEL
LIN {X 0,Y 455.319,Z 930.963,A -85,B 0,C 180,E1 8028.379,E2 8028.379} C_VEL
LIN {X 0,Y 458.111,Z 907.328,A -85,B 0,C 180,E1 8032.338,E2 8032.338} C_VEL
LIN {X 0,Y 461.613,Z 879.341,A -85,B 0,C 180,E1 8035.786,E2 8035.786} C_VEL
LIN {X 0,Y 465.375,Z 846.56,A -85,B 0,C 180,E1 8038.695,E2 8038.695} C_VEL
LIN {X 0,Y 468.685,Z 812.691,A -85,B 0,C 180,E1 8040.786,E2 8040.786} C_VEL
LIN {X 0,Y 470.335,Z 778.298,A -85,B 0,C 180,E1 8042.225,E2 8042.225} C_VEL
LIN {X 0,Y 454.454,Z 742.197,A -85,B 0,C 180,E1 8044.441,E2 8044.441} C_VEL
LIN {X 0,Y 450.945,Z 733.66,A -85,B 0,C 180,E1 8045.008,E2 8045.008} C_VEL
LIN {X 0,Y 450.818,Z 733.66,A -85,B 0,C 180,E1 8049.652,E2 8049.652} C_VEL
LIN {X 0,Y 450.803,Z 733.66,A -85,B 0,C 180,E1 8055.142,E2 8055.142} C_VEL
LIN {X 0,Y 450.878,Z 733.66,A -85,B 0,C 180,E1 8060.567,E2 8060.567} C_VEL
LIN {X 0,Y 450.852,Z 733.66,A -85,B 0,C 180,E1 8067.096,E2 8067.096} C_VEL
LIN {X 0,Y 451.16,Z 733.66,A -85,B 0,C 180,E1 8074.13,E2 8074.13} C_VEL
LIN {X 0,Y 451.353,Z 733.66,A -85,B 0,C 180,E1 8080.396,E2 8080.396} C_VEL
LIN {X 0,Y 451.347,Z 733.66,A -85,B 0,C 180,E1 8086.616,E2 8086.616} C_VEL
LIN {X 0,Y 451.657,Z 733.66,A -85,B 0,C 180,E1 8092.29,E2 8092.29} C_VEL
LIN {X 0,Y 451.977,Z 733.66,A -85,B 0,C 180,E1 8098.076,E2 8098.076} C_VEL
LIN {X 0,Y 451.891,Z 733.66,A -85,B 0,C 180,E1 8103.838,E2 8103.838} C_VEL
LIN {X 0,Y 451.617,Z 733.66,A -85,B 0,C 180,E1 8109.645,E2 8109.645} C_VEL
LIN {X 0,Y 451.391,Z 733.66,A -85,B 0,C 180,E1 8115.56,E2 8115.56} C_VEL
LIN {X 0,Y 451.233,Z 733.66,A -85,B 0,C 180,E1 8121.654,E2 8121.654} C_VEL
LIN {X 0,Y 451.008,Z 733.66,A -85,B 0,C 180,E1 8128.028,E2 8128.028} C_VEL
LIN {X 0,Y 450.861,Z 733.66,A -85,B 0,C 180,E1 8134.805,E2 8134.805} C_VEL
LIN {X 0,Y 450.852,Z 733.66,A -85,B 0,C 180,E1 8139.64,E2 8139.64} C_VEL
LIN {X 0,Y 450.858,Z 733.66,A -85,B 0,C 180,E1 8145.151,E2 8145.151} C_VEL
LIN {X 0,Y 450.907,Z 733.66,A -85,B 0,C 180,E1 8150.551,E2 8150.551} C_VEL
LIN {X 0,Y 450.963,Z 733.894,A -85,B 0,C 180,E1 8153.206,E2 8153.206} C_VEL
LIN {X 0,Y 458.599,Z 760.327,A -85,B 0,C 180,E1 8155.733,E2 8155.733} C_VEL
LIN {X 0,Y 470.791,Z 789.645,A -85,B 0,C 180,E1 8157.25,E2 8157.25} C_VEL
LIN {X 0,Y 469.008,Z 829.092,A -85,B 0,C 180,E1 8158.208,E2 8158.208} C_VEL
LIN {X 0,Y 468.755,Z 832.219,A -85,B 0,C 180,E1 8158.318,E2 8158.318} C_VEL
LIN {X 0,Y 467.173,Z 840.696,A -85,B 0,C 180,E1 8158.571,E2 8158.571} C_VEL
LIN {X 0,Y 459.538,Z 862.984,A -85,B 0,C 180,E1 8159.231,E2 8159.231} C_VEL
LIN {X 0,Y 459.276,Z 864.922,A -85,B 0,C 180,E1 8159.337,E2 8159.337} C_VEL
LIN {X 0,Y 455.766,Z 898.937,A -85,B 0,C 180,E1 8161.682,E2 8161.682} C_VEL
LIN {X 0,Y 451.958,Z 931.561,A -85,B 0,C 180,E1 8164.871,E2 8164.871} C_VEL
LIN {X 0,Y 448.772,Z 958.539,A -85,B 0,C 180,E1 8168.475,E2 8168.475} C_VEL
LIN {X 0,Y 446.396,Z 982.067,A -85,B 0,C 180,E1 8172.735,E2 8172.735} C_VEL
LIN {X 0,Y 445.074,Z 999.675,A -85,B 0,C 180,E1 8177.225,E2 8177.225} C_VEL
LIN {X 0,Y 444.592,Z 1011.188,A -85,B 0,C 180,E1 8181.54,E2 8181.54} C_VEL
LIN {X 0,Y 444.388,Z 1018.405,A -85,B 0,C 180,E1 8186.092,E2 8186.092} C_VEL
LIN {X 0,Y 444.348,Z 1020.319,A -85,B 0,C 180,E1 8190,E2 8190} C_VEL
LIN {X 0,Y 444.438,Z 1018.24,A -85,B 0,C 180,E1 8193.907,E2 8193.907} C_VEL
LIN {X 0,Y 444.641,Z 1011.131,A -85,B 0,C 180,E1 8198.465,E2 8198.465} C_VEL
LIN {X 0,Y 445.198,Z 998.063,A -85,B 0,C 180,E1 8203.271,E2 8203.271} C_VEL
LIN {X 0,Y 446.606,Z 979.621,A -85,B 0,C 180,E1 8207.765,E2 8207.765} C_VEL
LIN {X 0,Y 448.978,Z 956.917,A -85,B 0,C 180,E1 8211.774,E2 8211.774} C_VEL
LIN {X 0,Y 452.439,Z 927.959,A -85,B 0,C 180,E1 8215.538,E2 8215.538} C_VEL
LIN {X 0,Y 456.062,Z 897.096,A -85,B 0,C 180,E1 8218.459,E2 8218.459} C_VEL
LIN {X 0,Y 459.478,Z 864.139,A -85,B 0,C 180,E1 8220.701,E2 8220.701} C_VEL
LIN {X 0,Y 462.466,Z 826.813,A -85,B 0,C 180,E1 8222.378,E2 8222.378} C_VEL
LIN {X 0,Y 463.675,Z 789.076,A -85,B 0,C 180,E1 8223.325,E2 8223.325} C_VEL
LIN {X 0,Y 453.617,Z 762.384,A -85,B 0,C 180,E1 8224.657,E2 8224.657} C_VEL
LIN {X 0,Y 444.834,Z 738.669,A -85,B 0,C 180,E1 8225.896,E2 8225.896} C_VEL
LIN {X 0,Y 443.027,Z 733.66,A -85,B 0,C 180,E1 8226.224,E2 8226.224} C_VEL
LIN {X 0,Y 442.888,Z 733.66,A -85,B 0,C 180,E1 8233.136,E2 8233.136} C_VEL
LIN {X 0,Y 442.848,Z 733.66,A -85,B 0,C 180,E1 8239.496,E2 8239.496} C_VEL
LIN {X 0,Y 443.011,Z 733.66,A -85,B 0,C 180,E1 8245.11,E2 8245.11} C_VEL
LIN {X 0,Y 443.041,Z 733.66,A -85,B 0,C 180,E1 8251.423,E2 8251.423} C_VEL
LIN {X 0,Y 443.277,Z 734.265,A -85,B 0,C 180,E1 8255.226,E2 8255.226} C_VEL
LIN {X 0,Y 453.144,Z 763.648,A -85,B 0,C 180,E1 8256.896,E2 8256.896} C_VEL
LIN {X 0,Y 453.071,Z 793.081,A -85,B 0,C 180,E1 8258.009,E2 8258.009} C_VEL
LIN {X 0,Y 451.707,Z 819.9,A -85,B 0,C 180,E1 8259.807,E2 8259.807} C_VEL
LIN {X 0,Y 450.139,Z 842.327,A -85,B 0,C 180,E1 8262.131,E2 8262.131} C_VEL
LIN {X 0,Y 448.39,Z 861.466,A -85,B 0,C 180,E1 8265.085,E2 8265.085} C_VEL
LIN {X 0,Y 447.087,Z 875.168,A -85,B 0,C 180,E1 8268.281,E2 8268.281} C_VEL
LIN {X 0,Y 446.208,Z 883.13,A -85,B 0,C 180,E1 8271.222,E2 8271.222} C_VEL
LIN {X 0,Y 445.91,Z 887.354,A -85,B 0,C 180,E1 8274.158,E2 8274.158} C_VEL
LIN {X 0,Y 445.58,Z 887.803,A -85,B 0,C 180,E1 8278.057,E2 8278.057} C_VEL
LIN {X 0,Y 445.761,Z 882.321,A -85,B 0,C 180,E1 8281.951,E2 8281.951} C_VEL
LIN {X 0,Y 446.328,Z 872.259,A -85,B 0,C 180,E1 8285.357,E2 8285.357} C_VEL
LIN {X 0,Y 447.295,Z 856.053,A -85,B 0,C 180,E1 8288.766,E2 8288.766} C_VEL
LIN {X 0,Y 448.713,Z 835.223,A -85,B 0,C 180,E1 8291.684,E2 8291.684} C_VEL
LIN {X 0,Y 450.19,Z 810.916,A -85,B 0,C 180,E1 8293.992,E2 8293.992} C_VEL
LIN {X 0,Y 451.435,Z 782.202,A -85,B 0,C 180,E1 8295.738,E2 8295.738} C_VEL
LIN {X 0,Y 451.034,Z 760.758,A -85,B 0,C 180,E1 8296.557,E2 8296.557} C_VEL
LIN {X 0,Y 443.42,Z 733.66,A -85,B 0,C 180,E1 8297.56,E2 8297.56} C_VEL
LIN {X 0,Y 443.203,Z 733.66,A -85,B 0,C 180,E1 8304.205,E2 8304.205} C_VEL
LIN {X 0,Y 442.958,Z 733.66,A -85,B 0,C 180,E1 8311.292,E2 8311.292} C_VEL
LIN {X 0,Y 442.928,Z 733.66,A -85,B 0,C 180,E1 8315.533,E2 8315.533} C_VEL
LIN {X 0,Y 442.83,Z 733.66,A -85,B 0,C 180,E1 8321.218,E2 8321.218} C_VEL
LIN {X 0,Y 442.903,Z 733.66,A -85,B 0,C 180,E1 8326.866,E2 8326.866} C_VEL
LIN {X 0,Y 443.008,Z 733.66,A -85,B 0,C 180,E1 8334.016,E2 8334.016} C_VEL
LIN {X 0,Y 443.027,Z 733.717,A -85,B 0,C 180,E1 8334.268,E2 8334.268} C_VEL
LIN {X 0,Y 462.454,Z 777.821,A -85,B 0,C 180,E1 8337.033,E2 8337.033} C_VEL
LIN {X 0,Y 463.907,Z 786.082,A -85,B 0,C 180,E1 8337.458,E2 8337.458} C_VEL
LIN {X 0,Y 461.049,Z 822.255,A -85,B 0,C 180,E1 8339.112,E2 8339.112} C_VEL
LIN {X 0,Y 457.385,Z 856.059,A -85,B 0,C 180,E1 8341.459,E2 8341.459} C_VEL
LIN {X 0,Y 453.458,Z 887.352,A -85,B 0,C 180,E1 8344.529,E2 8344.529} C_VEL
LIN {X 0,Y 449.784,Z 914.836,A -85,B 0,C 180,E1 8348.267,E2 8348.267} C_VEL
LIN {X 0,Y 446.985,Z 937.546,A -85,B 0,C 180,E1 8352.505,E2 8352.505} C_VEL
LIN {X 0,Y 445.41,Z 953.772,A -85,B 0,C 180,E1 8356.735,E2 8356.735} C_VEL
LIN {X 0,Y 444.563,Z 966.036,A -85,B 0,C 180,E1 8361.553,E2 8361.553} C_VEL
LIN {X 0,Y 444.251,Z 972.416,A -85,B 0,C 180,E1 8366.092,E2 8366.092} C_VEL
LIN {X 0,Y 444.253,Z 974.158,A -85,B 0,C 180,E1 8370,E2 8370} C_VEL
LIN {X 0,Y 444.366,Z 971.348,A -85,B 0,C 180,E1 8374.887,E2 8374.887} C_VEL
LIN {X 0,Y 444.754,Z 962.969,A -85,B 0,C 180,E1 8379.801,E2 8379.801} C_VEL
LIN {X 0,Y 445.734,Z 949.99,A -85,B 0,C 180,E1 8384.294,E2 8384.294} C_VEL
LIN {X 0,Y 447.829,Z 930.893,A -85,B 0,C 180,E1 8388.792,E2 8388.792} C_VEL
LIN {X 0,Y 450.623,Z 908.521,A -85,B 0,C 180,E1 8392.609,E2 8392.609} C_VEL
LIN {X 0,Y 454.42,Z 879.966,A -85,B 0,C 180,E1 8396.198,E2 8396.198} C_VEL
LIN {X 0,Y 458.369,Z 847.501,A -85,B 0,C 180,E1 8399.13,E2 8399.13} C_VEL
LIN {X 0,Y 461.912,Z 812.925,A -85,B 0,C 180,E1 8401.296,E2 8401.296} C_VEL
LIN {X 0,Y 463.672,Z 780.99,A -85,B 0,C 180,E1 8402.658,E2 8402.658} C_VEL
LIN {X 0,Y 448.732,Z 746.46,A -85,B 0,C 180,E1 8404.867,E2 8404.867} C_VEL
LIN {X 0,Y 442.99,Z 733.66,A -85,B 0,C 180,E1 8405.704,E2 8405.704} C_VEL
LIN {X 0,Y 442.788,Z 733.66,A -85,B 0,C 180,E1 8413.149,E2 8413.149} C_VEL
LIN {X 0,Y 442.877,Z 733.66,A -85,B 0,C 180,E1 8419.488,E2 8419.488} C_VEL
LIN {X 0,Y 442.948,Z 733.66,A -85,B 0,C 180,E1 8425.123,E2 8425.123} C_VEL
LIN {X 0,Y 443.063,Z 733.66,A -85,B 0,C 180,E1 8431.414,E2 8431.414} C_VEL
LIN {X 0,Y 443.319,Z 733.66,A -85,B 0,C 180,E1 8437.93,E2 8437.93} C_VEL
LIN {X 0,Y 443.365,Z 733.66,A -85,B 0,C 180,E1 8444.142,E2 8444.142} C_VEL
LIN {X 0,Y 443.584,Z 733.66,A -85,B 0,C 180,E1 8450.17,E2 8450.17} C_VEL
LIN {X 0,Y 443.796,Z 733.66,A -85,B 0,C 180,E1 8456.083,E2 8456.083} C_VEL
LIN {X 0,Y 443.953,Z 733.66,A -85,B 0,C 180,E1 8461.95,E2 8461.95} C_VEL
LIN {X 0,Y 443.679,Z 733.66,A -85,B 0,C 180,E1 8468.248,E2 8468.248} C_VEL
LIN {X 0,Y 443.501,Z 733.66,A -85,B 0,C 180,E1 8473.821,E2 8473.821} C_VEL
LIN {X 0,Y 443.37,Z 733.66,A -85,B 0,C 180,E1 8479.962,E2 8479.962} C_VEL
LIN {X 0,Y 443.148,Z 733.66,A -85,B 0,C 180,E1 8486.364,E2 8486.364} C_VEL
LIN {X 0,Y 442.97,Z 733.66,A -85,B 0,C 180,E1 8493.146,E2 8493.146} C_VEL
LIN {X 0,Y 442.872,Z 733.66,A -85,B 0,C 180,E1 8498.156,E2 8498.156} C_VEL
LIN {X 0,Y 442.892,Z 733.66,A -85,B 0,C 180,E1 8504.117,E2 8504.117} C_VEL
LIN {X 0,Y 442.899,Z 733.66,A -85,B 0,C 180,E1 8509.493,E2 8509.493} C_VEL
LIN {X 0,Y 443.045,Z 733.949,A -85,B 0,C 180,E1 8512.643,E2 8512.643} C_VEL
LIN {X 0,Y 449.867,Z 757.394,A -85,B 0,C 180,E1 8514.923,E2 8514.923} C_VEL
LIN {X 0,Y 464.102,Z 791.028,A -85,B 0,C 180,E1 8516.746,E2 8516.746} C_VEL
LIN {X 0,Y 462.177,Z 830.139,A -85,B 0,C 180,E1 8517.741,E2 8517.741} C_VEL
LIN {X 0,Y 459.276,Z 864.922,A -85,B 0,C 180,E1 8519.337,E2 8519.337} C_VEL
LIN {X 0,Y 454.296,Z 880.812,A -85,B 0,C 180,E1 8520.087,E2 8520.087} C_VEL
LIN {X 0,Y 449.026,Z 895.823,A -85,B 0,C 180,E1 8520.976,E2 8520.976} C_VEL
LIN {X 0,Y 445.094,Z 927.616,A -85,B 0,C 180,E1 8524.017,E2 8524.017} C_VEL
LIN {X 0,Y 441.4,Z 956.507,A -85,B 0,C 180,E1 8527.832,E2 8527.832} C_VEL
LIN {X 0,Y 438.89,Z 979.211,A -85,B 0,C 180,E1 8531.911,E2 8531.911} C_VEL
LIN {X 0,Y 437.376,Z 997.654,A -85,B 0,C 180,E1 8536.486,E2 8536.486} C_VEL
LIN {X 0,Y 436.694,Z 1010.734,A -85,B 0,C 180,E1 8541.385,E2 8541.385} C_VEL
LIN {X 0,Y 436.546,Z 1017.615,A -85,B 0,C 180,E1 8546.022,E2 8546.022} C_VEL
LIN {X 0,Y 436.506,Z 1019.521,A -85,B 0,C 180,E1 8550,E2 8550} C_VEL
LIN {X 0,Y 436.615,Z 1016.583,A -85,B 0,C 180,E1 8554.973,E2 8554.973} C_VEL
LIN {X 0,Y 436.735,Z 1009.358,A -85,B 0,C 180,E1 8559.269,E2 8559.269} C_VEL
LIN {X 0,Y 437.482,Z 995.878,A -85,B 0,C 180,E1 8564.02,E2 8564.02} C_VEL
LIN {X 0,Y 439.073,Z 977.44,A -85,B 0,C 180,E1 8568.456,E2 8568.456} C_VEL
LIN {X 0,Y 441.771,Z 953.871,A -85,B 0,C 180,E1 8572.578,E2 8572.578} C_VEL
LIN {X 0,Y 445.375,Z 925.365,A -85,B 0,C 180,E1 8576.228,E2 8576.228} C_VEL
LIN {X 0,Y 449.307,Z 894.142,A -85,B 0,C 180,E1 8579.156,E2 8579.156} C_VEL
LIN {X 0,Y 453.086,Z 859.376,A -85,B 0,C 180,E1 8581.468,E2 8581.468} C_VEL
LIN {X 0,Y 456.128,Z 821.948,A -85,B 0,C 180,E1 8583.05,E2 8583.05} C_VEL
LIN {X 0,Y 456.995,Z 791.602,A -85,B 0,C 180,E1 8583.826,E2 8583.826} C_VEL
LIN {X 0,Y 446.804,Z 763.126,A -85,B 0,C 180,E1 8585.245,E2 8585.245} C_VEL
LIN {X 0,Y 438.825,Z 742.584,A -85,B 0,C 180,E1 8586.384,E2 8586.384} C_VEL
LIN {X 0,Y 435.128,Z 733.66,A -85,B 0,C 180,E1 8587.024,E2 8587.024} C_VEL
LIN {X 0,Y 435.006,Z 733.66,A -85,B 0,C 180,E1 8594.117,E2 8594.117} C_VEL
LIN {X 0,Y 434.903,Z 733.66,A -85,B 0,C 180,E1 8601.204,E2 8601.204} C_VEL
LIN {X 0,Y 435.092,Z 733.66,A -85,B 0,C 180,E1 8606.635,E2 8606.635} C_VEL
LIN {X 0,Y 435.225,Z 733.66,A -85,B 0,C 180,E1 8613.971,E2 8613.971} C_VEL
LIN {X 0,Y 435.317,Z 734.223,A -85,B 0,C 180,E1 8614.505,E2 8614.505} C_VEL
LIN {X 0,Y 445.128,Z 761.606,A -85,B 0,C 180,E1 8616.288,E2 8616.288} C_VEL
LIN {X 0,Y 446.474,Z 773.607,A -85,B 0,C 180,E1 8616.751,E2 8616.751} C_VEL
LIN {X 0,Y 445.588,Z 802.375,A -85,B 0,C 180,E1 8618.057,E2 8618.057} C_VEL
LIN {X 0,Y 444.079,Z 828.131,A -85,B 0,C 180,E1 8620.071,E2 8620.071} C_VEL
LIN {X 0,Y 442.244,Z 849.371,A -85,B 0,C 180,E1 8622.574,E2 8622.574} C_VEL
LIN {X 0,Y 440.365,Z 867.755,A -85,B 0,C 180,E1 8625.825,E2 8625.825} C_VEL
LIN {X 0,Y 439.007,Z 880.158,A -85,B 0,C 180,E1 8629.244,E2 8629.244} C_VEL
LIN {X 0,Y 438.199,Z 887.662,A -85,B 0,C 180,E1 8633.059,E2 8633.059} C_VEL
LIN {X 0,Y 437.86,Z 889.648,A -85,B 0,C 180,E1 8636.039,E2 8636.039} C_VEL
LIN {X 0,Y 437.819,Z 887.067,A -85,B 0,C 180,E1 8640.004,E2 8640.004} C_VEL
LIN {X 0,Y 438.275,Z 878.461,A -85,B 0,C 180,E1 8643.966,E2 8643.966} C_VEL
LIN {X 0,Y 439.177,Z 863.826,A -85,B 0,C 180,E1 8647.681,E2 8647.681} C_VEL
LIN {X 0,Y 440.447,Z 844.634,A -85,B 0,C 180,E1 8650.849,E2 8650.849} C_VEL
LIN {X 0,Y 442.038,Z 820.785,A -85,B 0,C 180,E1 8653.498,E2 8653.498} C_VEL
LIN {X 0,Y 443.541,Z 793.807,A -85,B 0,C 180,E1 8655.471,E2 8655.471} C_VEL
LIN {X 0,Y 444.021,Z 764.07,A -85,B 0,C 180,E1 8656.765,E2 8656.765} C_VEL
LIN {X 0,Y 435.489,Z 733.66,A -85,B 0,C 180,E1 8657.921,E2 8657.921} C_VEL
LIN {X 0,Y 435.23,Z 733.66,A -85,B 0,C 180,E1 8664.678,E2 8664.678} C_VEL
LIN {X 0,Y 435.056,Z 733.66,A -85,B 0,C 180,E1 8671.472,E2 8671.472} C_VEL
LIN {X 0,Y 434.899,Z 733.66,A -85,B 0,C 180,E1 8676.8,E2 8676.8} C_VEL
LIN {X 0,Y 434.93,Z 733.66,A -85,B 0,C 180,E1 8683.025,E2 8683.025} C_VEL
LIN {X 0,Y 435.001,Z 733.66,A -85,B 0,C 180,E1 8688.599,E2 8688.599} C_VEL
LIN {X 0,Y 435.082,Z 733.684,A -85,B 0,C 180,E1 8693.505,E2 8693.505} C_VEL
LIN {X 0,Y 443.793,Z 752.311,A -85,B 0,C 180,E1 8694.704,E2 8694.704} C_VEL
LIN {X 0,Y 457.197,Z 784.488,A -85,B 0,C 180,E1 8696.847,E2 8696.847} C_VEL
LIN {X 0,Y 454.297,Z 822.294,A -85,B 0,C 180,E1 8698.579,E2 8698.579} C_VEL
LIN {X 0,Y 450.493,Z 855.692,A -85,B 0,C 180,E1 8700.913,E2 8700.913} C_VEL
LIN {X 0,Y 446.396,Z 886.675,A -85,B 0,C 180,E1 8703.966,E2 8703.966} C_VEL
LIN {X 0,Y 442.543,Z 913.705,A -85,B 0,C 180,E1 8707.632,E2 8707.632} C_VEL
LIN {X 0,Y 439.503,Z 936.778,A -85,B 0,C 180,E1 8711.938,E2 8711.938} C_VEL
LIN {X 0,Y 437.672,Z 954.175,A -85,B 0,C 180,E1 8716.496,E2 8716.496} C_VEL
LIN {X 0,Y 436.733,Z 966.44,A -85,B 0,C 180,E1 8721.401,E2 8721.401} C_VEL
LIN {X 0,Y 436.365,Z 972.822,A -85,B 0,C 180,E1 8726.021,E2 8726.021} C_VEL
LIN {X 0,Y 436.391,Z 974.563,A -85,B 0,C 180,E1 8730,E2 8730} C_VEL
LIN {X 0,Y 436.486,Z 971.756,A -85,B 0,C 180,E1 8734.975,E2 8734.975} C_VEL
LIN {X 0,Y 436.918,Z 963.378,A -85,B 0,C 180,E1 8739.978,E2 8739.978} C_VEL
LIN {X 0,Y 438.09,Z 949.721,A -85,B 0,C 180,E1 8744.754,E2 8744.754} C_VEL
LIN {X 0,Y 440.399,Z 930.084,A -85,B 0,C 180,E1 8749.368,E2 8749.368} C_VEL
LIN {X 0,Y 443.756,Z 905.767,A -85,B 0,C 180,E1 8753.471,E2 8753.471} C_VEL
LIN {X 0,Y 447.742,Z 876.794,A -85,B 0,C 180,E1 8757.027,E2 8757.027} C_VEL
LIN {X 0,Y 451.769,Z 845.099,A -85,B 0,C 180,E1 8759.831,E2 8759.831} C_VEL
LIN {X 0,Y 455.486,Z 809.821,A -85,B 0,C 180,E1 8761.997,E2 8761.997} C_VEL
LIN {X 0,Y 456.93,Z 783.406,A -85,B 0,C 180,E1 8763.124,E2 8763.124} C_VEL
LIN {X 0,Y 442.087,Z 748.665,A -85,B 0,C 180,E1 8765.431,E2 8765.431} C_VEL
LIN {X 0,Y 435.06,Z 733.66,A -85,B 0,C 180,E1 8766.428,E2 8766.428} C_VEL
LIN {X 0,Y 434.872,Z 733.66,A -85,B 0,C 180,E1 8773.013,E2 8773.013} C_VEL
LIN {X 0,Y 434.957,Z 733.66,A -85,B 0,C 180,E1 8778.591,E2 8778.591} C_VEL
LIN {X 0,Y 434.934,Z 733.66,A -85,B 0,C 180,E1 8783.712,E2 8783.712} C_VEL
LIN {X 0,Y 435.042,Z 733.66,A -85,B 0,C 180,E1 8788.527,E2 8788.527} C_VEL
LIN {X 0,Y 435.284,Z 733.66,A -85,B 0,C 180,E1 8795.325,E2 8795.325} C_VEL
LIN {X 0,Y 435.498,Z 733.66,A -85,B 0,C 180,E1 8801.762,E2 8801.762} C_VEL
LIN {X 0,Y 435.517,Z 733.66,A -85,B 0,C 180,E1 8807.956,E2 8807.956} C_VEL
LIN {X 0,Y 435.906,Z 733.66,A -85,B 0,C 180,E1 8814.015,E2 8814.015} C_VEL
LIN {X 0,Y 436.16,Z 733.66,A -85,B 0,C 180,E1 8819.996,E2 8819.996} C_VEL
LIN {X 0,Y 435.844,Z 733.66,A -85,B 0,C 180,E1 8825.977,E2 8825.977} C_VEL
LIN {X 0,Y 435.635,Z 733.66,A -85,B 0,C 180,E1 8832.031,E2 8832.031} C_VEL
LIN {X 0,Y 435.474,Z 733.66,A -85,B 0,C 180,E1 8838.229,E2 8838.229} C_VEL
LIN {X 0,Y 435.211,Z 733.66,A -85,B 0,C 180,E1 8845.238,E2 8845.238} C_VEL
LIN {X 0,Y 435.066,Z 733.66,A -85,B 0,C 180,E1 8851.461,E2 8851.461} C_VEL
LIN {X 0,Y 434.905,Z 733.66,A -85,B 0,C 180,E1 8856.8,E2 8856.8} C_VEL
LIN {X 0,Y 434.943,Z 733.66,A -85,B 0,C 180,E1 8863.026,E2 8863.026} C_VEL
LIN {X 0,Y 434.986,Z 733.66,A -85,B 0,C 180,E1 8868.597,E2 8868.597} C_VEL
LIN {X 0,Y 435.052,Z 733.702,A -85,B 0,C 180,E1 8872.041,E2 8872.041} C_VEL
LIN {X 0,Y 441.198,Z 754.348,A -85,B 0,C 180,E1 8874.076,E2 8874.076} C_VEL
LIN {X 0,Y 457.435,Z 795.617,A -85,B 0,C 180,E1 8876.299,E2 8876.299} C_VEL
LIN {X 0,Y 455.198,Z 832.739,A -85,B 0,C 180,E1 8877.312,E2 8877.312} C_VEL
LIN {X 0,Y 451.934,Z 869.778,A -85,B 0,C 180,E1 8879.125,E2 8879.125} C_VEL
LIN {X 0,Y 449.026,Z 895.823,A -85,B 0,C 180,E1 8880.976,E2 8880.976} C_VEL
LIN {X 0,Y 443.671,Z 910.509,A -85,B 0,C 180,E1 8882.028,E2 8882.028} C_VEL
LIN {X 0,Y 438.262,Z 924.239,A -85,B 0,C 180,E1 8883.228,E2 8883.228} C_VEL
LIN {X 0,Y 434.33,Z 952.792,A -85,B 0,C 180,E1 8886.909,E2 8886.909} C_VEL
LIN {X 0,Y 431.432,Z 976.304,A -85,B 0,C 180,E1 8891.047,E2 8891.047} C_VEL
